Logger.s1:=CONCAT(Logger.s1,DINT_TO_STRING(measures.COSPHI_L1));		Logger.s1:=CONCAT(Logger.s1,';');
Logger.s1:=CONCAT(Logger.s1,DINT_TO_STRING(measures.COSPHI_L2));		Logger.s1:=CONCAT(Logger.s1,';');
Logger.s1:=CONCAT(Logger.s1,DINT_TO_STRING(measures.COSPHI_L3));		Logger.s1:=CONCAT(Logger.s1,';');

Logger.s1:=CONCAT(Logger.s1,BYTE_TO_STRING(SEL(contabilizerMode=THREE_PHASE,1,0)));

ADDSTRING(ADR(Logger.TData), ADR(Logger.s1), Logger.TLen);*)
;
END_ACTION
ACTION checkAlarm:
(*IF(alarmLaunched[1]=0 AND typ_750_494_State.xPhase1_OverCurrentSystem) THEN
	alarmLaunched[1]:=2;
	LogEv(EL_Alarm,EO_ANZ,ID,3, 'xPhase1_OverCurrentSystem');
ELSIF (alarmLaunched[1]=2 AND NOT(typ_750_494_State.xPhase1_OverCurrentSystem) ) THEN
	alarmLaunched[1]:=0;
	LogEv(EL_Log,EO_ANZ,ID,4,'xPhase1_OverCurrentSystem');
END_IF*)

;
END_ACTION
ACTION checkEventsToSignal:
CheckAlarm();
CheckWarning();
CheckStatus();
END_ACTION
ACTION checkStatus:
(*tmpAlarm:=0;
FOR I:=1 TO MAX_alarm DO tmpAlarm:=tmpAlarm+alarmLaunched[i]; END_FOR
IF(tmpAlarm>0) THEN status_Log:=2; END_IF

tmpWarning:=0;
FOR I:=1 TO MAX_WARNING DO tmpWarning:=tmpWarning+warningLaunched[i]; END_FOR
IF(status=0 AND tmpWarning>0) THEN status:=1; END_IF

IF (tmpAlarm =0 AND tmpWarning =0) THEN status:=0; END_IF*)
;
END_ACTION
ACTION checkWarning:
IF(enableWarning = FALSE) THEN RETURN; END_IF

(*IF( warningLaunched[1]=0 AND typ_750_494_State.xGeneralError) THEN
	warningLaunched[1]:=2;
	LogEv(EL_Wrn,EO_ANZ,ID,5, 'xGeneralError');
ELSIF (warningLaunched[1]=2 AND NOT(typ_750_494_State.xGeneralError) ) THEN
	warningLaunched[1]:=0;
	LogEv(EL_Log,EO_ANZ,ID,5,'xGeneralError');
END_IF*)

;
END_ACTION
ACTION convertToClevergyFormat:
	measures.V_L1N := specificData.arVoltage_L_N[1];
	measures.V_L2N := specificData.arVoltage_L_N[2];
	measures.V_L3N := specificData.arVoltage_L_N[3];

	(*n/a*)
	measures.V_L1L2:=0;
	measures.V_L2L3:=0;
	measures.V_L3L1:=0;

	measures.FREQ := specificData.arFrequency*1000;

	measures.I_L1 := specificData.arCurrent[1]*1000;
	measures.I_L2 := specificData.arCurrent[2]*1000;
	measures.I_L3 :=specificData.arCurrent[3]*1000;

	measures.I_L1_Max := specificData.rMaximumCurrentL1*1000;
	measures.I_L2_Max := specificData.rMaximumCurrentL2*1000;
	measures.I_L3_Max := specificData.rMaximumCurrentL3*1000;

	measures.PF_L1 := specificData.arPowerFactorPF[1]*1000;
	measures.PF_L2 := specificData.arPowerFactorPF[2]*1000;
	measures.PF_L3 := specificData.arPowerFactorPF[3]*1000;

	measures.P_3P := specificData.rTotalActivePower*1000;
	measures.P_3P_Avg:=specificData.rAverageTotalActivePower*1000;
	measures.P_3P_Max:=specificData.rMaximumTotalActivePower*1000;

	measures.Q_3P:=specificData.rTotalReactivePower*1000;
	measures.Q_3P_Max:=specificData.rMaximumTotalReactivePower*1000;

	measures.WH_3P:=specificData.rTotalActiveEnergy*10;
	measures.VARH_3P:=specificData.rTotalReactiveEnergy*10;

	(*n/a*)
	measures.COSPHI_L1:=0;
	measures.COSPHI_L2:=0;
	measures.COSPHI_L3:=0;
END_ACTION
ACTION convertToClevergyFormat_OLD:
	measures.V_L1N := REAL_TO_DWORD(specificData.arVoltage_L_N[1]);
	measures.V_L2N := REAL_TO_DWORD(specificData.arVoltage_L_N[2]);
	measures.V_L3N := REAL_TO_DWORD(specificData.arVoltage_L_N[3]);

	(*n/a*)
	measures.V_L1L2:=REAL_TO_DWORD(0);
	measures.V_L2L3:=REAL_TO_DWORD(0);
	measures.V_L3L1:=REAL_TO_DWORD(0);

	measures.FREQ := REAL_TO_DWORD(specificData.arFrequency*1000);

	measures.I_L1 := REAL_TO_DWORD(specificData.arCurrent[1]*1000);
	measures.I_L2 := REAL_TO_DWORD(specificData.arCurrent[2]*1000);
	measures.I_L3 := REAL_TO_DWORD(specificData.arCurrent[3]*1000);

	measures.I_L1_Max := REAL_TO_DWORD(specificData.rMaximumCurrentL1*1000);
	measures.I_L2_Max := REAL_TO_DWORD(specificData.rMaximumCurrentL2*1000);
	measures.I_L3_Max := REAL_TO_DWORD(specificData.rMaximumCurrentL3*1000);

	measures.PF_L1 := REAL_TO_DINT(specificData.arPowerFactorPF[1]*1000);
	measures.PF_L2 := REAL_TO_DINT(specificData.arPowerFactorPF[2]*1000);
	measures.PF_L3 := REAL_TO_DINT(specificData.arPowerFactorPF[3]*1000);

	measures.P_3P := REAL_TO_DINT(specificData.rTotalActivePower);
	measures.P_3P_Avg:=REAL_TO_DINT(specificData.rAverageTotalActivePower);
	measures.P_3P_Max:=REAL_TO_DINT(specificData.rMaximumTotalActivePower);

	measures.Q_3P:=REAL_TO_DINT(specificData.rTotalReactivePower);
	measures.Q_3P_Max:=REAL_TO_DINT(specificData.rMaximumTotalReactivePower);

	measures.WH_3P:=REAL_TO_DINT(specificData.rTotalActiveEnergy*10);
	measures.VARH_3P:=REAL_TO_DINT(specificData.rTotalReactiveEnergy*10);

	(*n/a*)
	measures.COSPHI_L1:=REAL_TO_DINT(0);
	measures.COSPHI_L2:=REAL_TO_DINT(0);
	measures.COSPHI_L3:=REAL_TO_DINT(0);
;
END_ACTION
ACTION getModbusData:
specificData.arFrequency:=modBusConnector.regData[4];

specificData.arVoltage_L_N[1]:=modBusConnector.regData[1];
specificData.arVoltage_L_N[2]:=modBusConnector.regData[2];
specificData.arVoltage_L_N[3]:=modBusConnector.regData[3];

specificData.arCurrent[1]:=modBusConnector.regData[5];
specificData.arCurrent[2]:=modBusConnector.regData[6];
specificData.arCurrent[3]:=modBusConnector.regData[7];

specificData.rTotalActivePower:=modBusConnector.regData[8];
specificData.arActivePower[1]:=modBusConnector.regData[9];
specificData.arActivePower[2]:=modBusConnector.regData[10];
specificData.arActivePower[3]:=modBusConnector.regData[11];

specificData.rTotalReactivePower:=modBusConnector.regData[12];
specificData.arReactivePower[1]:=modBusConnector.regData[13];
specificData.arReactivePower[2]:=modBusConnector.regData[14];
specificData.arReactivePower[3]:=modBusConnector.regData[15];

specificData.rTotalApparentPower:=modBusConnector.regData[16];
specificData.arApparentPower[1]:=modBusConnector.regData[17];
specificData.arApparentPower[2]:=modBusConnector.regData[18];
specificData.arApparentPower[3]:=modBusConnector.regData[19];

specificData.rTotalPowerFactorPF:=modBusConnector.regData[20];
specificData.arPowerFactorPF[1]:=modBusConnector.regData[21];
specificData.arPowerFactorPF[2]:=modBusConnector.regData[22];
specificData.arPowerFactorPF[3]:=modBusConnector.regData[23];

specificData.rTotalActiveEnergy:=modBusConnector.regData[24];

specificData.rTotalReactiveEnergy:=modBusConnector.regData[25];
END_ACTION

(* POU ClevergyBlocks/OBJ_ANZ_INEPRO_PRO380/obj_MODBUS_GENERIC_CONNECTOR, ST *)
FUNCTION_BLOCK obj_MODBUS_GENERIC_CONNECTOR
VAR CONSTANT
		(* States of normal modbus data reading *)
		WAIT_STATE			:	BYTE := 0;
		QUERY_START_CYCLE	: 	BYTE := 1;
		QUERY_MEAS_REQ		:  	BYTE := 2;
		QUERY_MEAS_ANSW	: 	BYTE := 3;
		ERROR_STATE			:	BYTE := 4;
END_VAR
VAR_INPUT
		PARENT_EO_TYPE 		: 	WORD;
		PARENT_EO_ID		:	BYTE;
		Address				:	BYTE;
		TIMING				:	TIME:=t#500ms;

		retryErrMax			:	BYTE := 10;

END_VAR
VAR_IN_OUT
		ModBus		:	obj_MODBUS_ANZ;
END_VAR
VAR_OUTPUT
		Status_Log	:	BYTE;
		Status_Vis	:	DWORD;

		regDescr : ARRAY[1..MODBUS_INEPRO_MAX_REG] OF STRING(20);
		regAddress : ARRAY[1..MODBUS_INEPRO_MAX_REG] OF WORD;
		regQuantity : ARRAY[1..MODBUS_INEPRO_MAX_REG] OF BYTE;
		regValueType : ARRAY[1..MODBUS_INEPRO_MAX_REG] OF en_Modbus_Reg_Type;
		regData: ARRAY[1..MODBUS_INEPRO_MAX_REG] OF REAL;
		regDataWord: ARRAY[1..MODBUS_INEPRO_MAX_REG, 1..2] OF WORD;

END_VAR
VAR
		InitOK		:	BOOL := FALSE;

		(* Modbus State machine variables	*)
		state		:	BYTE;
		last_state		:	BYTE;
		retry		:	BYTE;
		retryErr		:	BYTE;
		ReadTmr		:	TON := (PT:=t#5s);	(* Just to do a first ModBus read at the beginning *)
		fModbusAlr	:	BOOL;

		(* Event check variable	*)
		Alarm		:	FLT_EVENT;
		ModBusAlr	:	FLT_EVENT := (INITEV:=FALSE);
		StatusOK		:	FLT_EVENT := (INITEV:=FALSE);
		AlarmCtr		:	BYTE;
		WarningCtr	:	BYTE;

		fTimeout	:	BOOL;

		currentReg:INT:=1;

		i:INT;
		x:INT;
END_VAR
IF NOT InitOK THEN
	ReadTmr.PT := timing;
	InitOK := TRUE;
	initMapping();
END_IF

(* State machine *)
Stm();

(* Check if an alarm has occured *)
CheckAlarm();

(* Set "Status_Log" according to actual object status	*)
IF AlarmCtr > 0 THEN
	Status_Log := 2;
	Status_Vis := COLOR_RED;
ELSIF WarningCtr > 0 THEN
	Status_Log := 1;
	Status_Vis := COLOR_YELLOW;
ELSE
	Status_Log := 0;

	Status_Vis := COLOR_GREEN;
END_IF
END_FUNCTION_BLOCK
ACTION CheckAlarm:
(*** Verify ModBus error	***)
ModbusAlr(IN:=fModbusAlr);

IF ModbusAlr.EVH THEN
	LogEv(EL_Alarm,PARENT_EO_TYPE,PARENT_EO_ID,2,SEL(ModBus.MB_MASTER.MB_Error<>0,'0','1'));
	AlarmCtr := AlarmCtr + 1;
END_IF

IF ModbusAlr.EVL THEN
	LogEv(EL_Log,PARENT_EO_TYPE,PARENT_EO_ID,1,'');
	AlarmCtr := SEL(AlarmCtr=0, AlarmCtr-1, 0);
END_IF
END_ACTION
ACTION initMapping:
FOR I:=1 TO MODBUS_INEPRO_MAX_REG DO

	IF MODBUS_INEPRO_RegAddress[PARENT_EO_ID,i] <> 0 THEN

		regAddress[i]:=MODBUS_INEPRO_RegAddress[PARENT_EO_ID, i];
		REGDescr[i]:=MODBUS_INEPRO_REGDescr[PARENT_EO_ID, i];
		regQuantity[i]:=MODBUS_INEPRO_regQuantity[PARENT_EO_ID, i];
		regValueType[i]:=MODBUS_INEPRO_regValueType[PARENT_EO_ID, i];

	END_IF

END_FOR
END_ACTION
ACTION Stm:
CASE state OF

	WAIT_STATE:	(* Refresh time manager *)

		ReadTmr(IN:=NOT(ReadTmr.Q));
		IF ReadTmr.Q THEN

			ReadTmr.PT := timing;			(* Refresh timer range *)

			(* Reset state machine variables and counters *)
			retry	:= 0;
			last_state	:= WAIT_STATE;

			(* Start state machine	*)
			state := QUERY_START_CYCLE;

		END_IF

	QUERY_START_CYCLE:
		IF NOT ModBus.MB_Start AND (NOT ModBus.MB_Lock OR retry>0) THEN
			ModBus.MB_Lock := TRUE;

			ModBus.MB_Obj := PARENT_EO_TYPE;
			ModBus.MB_ObjId := PARENT_EO_ID;

			state := QUERY_MEAS_REQ;
		END_IF

	(****			 MEASUREMENTS			  ****)

	QUERY_MEAS_REQ:
		IF NOT ModBus.MB_Start THEN

				IF regAddress[currentReg] <> 0 THEN

					ModBus.MB_Query.SlaveAddress := Address;
					ModBus.MB_Query.FunctionCode := 16#3;
					ModBus.MB_Query.Read_StartAddress :=regAddress[currentReg];
					ModBus.MB_Query.Read_Quantity := regQuantity[currentReg];
					ModBus.MB_Start := TRUE;

					state := QUERY_MEAS_ANSW;

				ELSE

					currentReg:=currentReg+1;

					IF(currentReg<=MODBUS_INEPRO_MAX_REG) THEN

						state := QUERY_MEAS_REQ;

					ELSE

						currentReg:=1;
						fModbusAlr := FALSE;
						retryErr := 0;
						ModBus.MB_Lock := FALSE;
						fTimeout := FALSE;
						state := WAIT_STATE;

					END_IF

				END_IF
		END_IF


	QUERY_MEAS_ANSW:
		IF NOT ModBus.MB_Start THEN
			IF ModBus.MB_MASTER.bInterfaceError<>0 OR ModBus.MB_MASTER.MB_Error<>0 THEN
				last_state := QUERY_MEAS_ANSW;
				state := ERROR_STATE;
			ELSE

				IF (regValueType[currentReg] = VALUE_REAL ) THEN
					regData[currentReg]:=BUILD_REAL_COPY(ModBus.MB_Resp.Data[1],ModBus.MB_Resp.Data[0]);
				END_IF
				IF (regValueType[currentReg] = VALUE_LONG ) THEN
					regDataWord[currentReg,1]:=ModBus.MB_Resp.Data[0];
					regDataWord[currentReg,2]:=ModBus.MB_Resp.Data[1];
				END_IF

				currentReg:=currentReg+1;

				IF(currentReg<=MODBUS_INEPRO_MAX_REG) THEN

					state := QUERY_MEAS_REQ;

				ELSE
					currentReg:=1;
					fModbusAlr := FALSE;
					retryErr := 0;
					ModBus.MB_Lock := FALSE;
					fTimeout := FALSE;
					state := WAIT_STATE;
				END_IF


			END_IF
		END_IF


	ERROR_STATE:	(* Error state *)

		IF retry < 3 THEN
			retry := retry+1;
			state := last_state;

		ELSE
			ModBus.MB_Lock := FALSE;

			(* Verify if slave is dead *)
			IF retryErr < retryErrMaX THEN
				retryErr := retryErr + 1;
			ELSE
				fModbusAlr := TRUE;
			END_IF

			(* Back to wait state *)
			state := WAIT_STATE;

			fTimeout := TRUE;
		END_IF

		IF ModBus.MB_MASTER.MB_Error=MB_TIME_OUT THEN
			state := state;
		END_IF
ELSE
	state := WAIT_STATE;
END_CASE
END_ACTION

(* POU ClevergyBlocks/obj_MODBUS_ANZ, ST *)
FUNCTION_BLOCK obj_MODBUS_ANZ
(* === MODBUS PROTOCOL INTERFACE ===
   v1.1[19/06/15] - Added new VARS allocation and searching
*)
VAR CONSTANT
	VARS_Max	: BYTE := 32;
END_VAR
VAR_INPUT
	(* Settings *)
	ID			: BYTE;
	COM			: BYTE;
	BAUDRATE	: COM_BAUDRATE;
	RS485		: BOOL := FALSE;
	PARITY : COM_PARITY:=PARITY_NO;
	STOP_BITS :COM_STOPBITS:=STOPBITS_2;
	TIME_OUT_TIME : TIME:=t#500ms;

	(* Interface *)
	MB_MASTER	: MODBUS_EXTENDED_MASTER;
	MB_Start	: BOOL;
	MB_Query	: typModbusExtendedQuery;
	MB_Resp		: typModbusResponse;
	MB_Lock		: BOOL;
	MB_Obj		: en_SYS_Objects;
	MB_ObjId	: BYTE;

	(* Variables management *)
	VARS_En		: BOOL := FALSE;
	VARS		: ARRAY [0..VARS_Max] OF typ_MODBUS_VAR_anz;
	VARS_Check	: BOOL;
	VARS_Alarm	: BOOL;

	(* Variables allocation *)
	VAR_Pointer : POINTER TO ARRAY[0..99] OF WORD;
	VAR_Cfg		: POINTER TO typ_MODBUS_VAR_ANZ;
END_VAR
VAR_OUTPUT
	(* Status *)
	Status_Log	: BYTE;
	Status_Vis	: DWORD;
END_VAR
VAR
	sta         : BYTE :=0;
	i			: BYTE;
	j			: BYTE;

	AlarmCOM	: FLT_EVENT;	(* Physical error relative to serial port -> COM	*)
	AlarmMDB	: FLT_EVENT;	(* ModBus error due to communication protocol error	*)

	VarTmr		: TON := (PT:=T#1s);
	VarSta		: BYTE; (* Status *)
	VarCnt		: BYTE; (* Scan counter *)
	VarRetry	: BYTE;
	VarAlarm	: BYTE; (* Last variable with errors *)
END_VAR
MB_MASTER(ENABLE:=TRUE,	ASCII_Mode:=FALSE, bCOM_PORT:=COM, cbCOM_BAUDRATE:=BAUDRATE, cpCOM_PARITY:=PARITY,
		csCOM_STOPBITS:=STOP_BITS,	cbsCOM_BYTESIZE:=BS_8, cfCOM_FLOW_CONTROL:=SEL(RS485,NO_FLOW_CONTROL,HALFDUPLEX),
		tTIME_OUT:=TIME_OUT_TIME,	StartFunction:=MB_Start, ExtQuery:=MB_Query, Response:=MB_Resp);

(* Process variable management *)
IF VARS_En THEN VARS_Process(); END_IF

(* Check status *)
AlarmCOM(IN:=(MB_MASTER.bInterfaceError<>0));
IF AlarmCOM.EVH THEN
	LogEv(SEL(MB_MASTER.bInterfaceError<>3,EL_Wrn,EL_Alarm),EO_MODBUS,ID,1,BYTE_TO_STRING(MB_MASTER.bInterfaceError));
END_IF
IF AlarmCOM.EVL THEN								(* Trigger a fall edge: MODBUS back working *)
	LogEv(EL_Log,EO_MODBUS,ID,2,'MODBUS_OK');
END_IF

(* If VARS not active check if a protocol error has occured (if VARS active this check is already done in "VARS_Process"	*)
IF NOT VARS_En THEN

	AlarmMDB(IN:=(MB_MASTER.MB_Error<>0));
(*	IF AlarmMDB.EVH THEN
		LogEv(EL_Wrn,EO_MODBUS,ID,2,INT_TO_STRING(MB_MASTER.MB_Error));
	END_IF
	IF AlarmMDB.EVL THEN								(* Trigger a fall edge: MODBUS back working *)
		LogEv(EL_Log,EO_MODBUS,ID,2,'MODBUS_OK');
	END_IF
*)
END_IF

(* Log/visu status *)
IF AlarmCOM.IN THEN Status_Log:=2; Status_Vis:=COLOR_RED;
ELSIF Vars_Alarm OR AlarmMDB.IN THEN Status_Log:=1; Status_Vis:=COLOR_YELLOW;
ELSE Status_Log:=0; Status_Vis:=COLOR_GREEN;
END_IF
END_FUNCTION_BLOCK
ACTION VAR_Search:
(* Search VAR with specific pointer if not found return first free VAR
	[Last VAR is not active... used as safe area...] 
*)
j:=VARS_Max;
FOR i := 0 TO VARS_Max-1 DO
	IF VARS[i].Variable=0 AND j>i THEN j:=i; END_IF
	IF VARS[i].Variable=VAR_Pointer THEN
		VAR_Cfg:=ADR(VARS[i]);
		RETURN;
	END_IF
END_FOR
VAR_Cfg:=ADR(VARS[j]);
END_ACTION
ACTION VARS_Process:
(* Update var timers *)
VarTmr(IN:=(NOT VarTmr.Q));
IF VarTmr.Q THEN
	FOR i := 0 TO VARS_Max DO
		IF VARS[i].Refresh_Cnt>0 THEN VARS[i].Refresh_Cnt:=VARS[i].Refresh_Cnt-1; END_IF
	END_FOR
	VARS_Check:=TRUE;
END_IF


(* Process status *)
CASE VarSta OF
	0: (* === Init *)
		VarCnt:=0;
		VarSta:=1;

	1: (* === Wait check signal *)
		IF VARS_Check THEN				(* Decremented "Refresh_Cnt" *)
			VARS_Check:=FALSE;
			VarCnt:=0;
			VarSta:=2;
		END_IF

	2: (* === Check loop *)
		IF NOT (MB_Lock OR MB_Start) THEN
			WHILE VarCnt<=(VARS_Max-1) AND VarSta=2 DO
				(* Check only active vars *)
				IF VARS[VarCnt].Variable<>0 THEN			(* "Variable" is a pointer to word, so if 0 no address *)
					(* Check var auto-refresh on timer checks *)
					IF VARS[VarCnt].Refresh_Time>0 AND VARS[VarCnt].Refresh_Cnt=0 THEN
						VARS[VarCnt].Refresh_Cnt:=VARS[VarCnt].Refresh_Time;
						VarSta:=3;
					END_IF
					(* Check refresh for change or request *)
					CASE VARS[VarCnt].FunCode OF
						5,6,15,16: (* Write functions *)
							IF VARS[VarCnt].Variable_Size=1 THEN
								IF VARS[VarCnt].Variable^[0]<>VARS[VarCnt].Variable_Mirror THEN
									VARS[VarCnt].Variable_Mirror:=VARS[VarCnt].Variable^[0];
									VarSta:=3;
								END_IF
							ELSE
								IF VARS[VarCnt].Variable_Mirror<>0 THEN
									VARS[VarCnt].Variable_Mirror:=0;
									VarSta:=3;
								END_IF
							END_IF
						1,2,3,4: (* Read functions *)
							IF VARS[VarCnt].Variable_Mirror<>0 THEN
								VARS[VarCnt].Variable_Mirror:=0;
								VarSta:=3;
							END_IF
					END_CASE
				END_IF
				(* Process query *)
				IF VarSta=3 THEN
					MB_Lock:=TRUE;
					MB_Query.SlaveAddress:=VARS[VarCnt].SlaveAddress;
					MB_Query.FunctionCode:=VARS[VarCnt].FunCode;
					CASE VARS[VarCnt].FunCode OF
						16#5,16#6,16#F,16#10:
							MB_Query.Read_Quantity:=0;
							MB_Query.Read_StartAddress:=0;
							MB_Query.Write_StartAddress:=VARS[VarCnt].FunAddress;
							MB_Query.Write_Quantity:=VARS[VarCnt].Variable_Size;
							IF VARS[VarCnt].Variable_Size=200 THEN
								COPY_32SWAP16(VARS[VarCnt].Variable, ADR(MB_Query.Write_Data[0]));
							ELSIF VARS[VarCnt].Variable_Size>1 THEN
								MEMCPY(VARS[VarCnt].Variable, ADR(MB_Query.Write_Data[0]), 2*VARS[VarCnt].Variable_Size);
							ELSE
								MB_Query.Write_Data[0]:=VARS[VarCnt].Variable^[0];
							END_IF
						16#1,16#2,16#3,16#4:
							MB_Query.Read_StartAddress:=VARS[VarCnt].FunAddress;
							IF VARS[VarCnt].Variable_Size=200 THEN MB_Query.Read_Quantity:=2; ELSE
							  MB_Query.Read_Quantity:=VARS[VarCnt].Variable_Size;
							END_IF
							MB_Query.Write_StartAddress:=0;
							MB_Query.Write_Quantity:=0;
					END_CASE
					VarRetry:=0;
					MB_Start:=TRUE;
				ELSE
					VarCnt:=VarCnt+1;
				END_IF
			END_WHILE
			(* Check loop completed -> no actions *)
			IF VarSta=2 THEN VarSta:=1; END_IF
		END_IF

	3: (* === Wait & process MB response *)
		IF NOT MB_Start THEN
			IF MB_MASTER.MB_Error=0 THEN
				CASE VARS[VarCnt].FunCode OF
					1,2,3,4:
						IF VARS[VarCnt].Variable_Size=200 THEN
							COPY_32SWAP16(ADR(MB_Resp.Data), VARS[VarCnt].Variable);
						ELSIF VARS[VarCnt].Variable_Size>1 THEN
							MEMCPY(ADR(MB_Resp.Data), VARS[VarCnt].Variable, 2*VARS[VarCnt].Variable_Size);
						ELSE
							VARS[VarCnt].Variable^[0]:=MB_Resp.Data[0];
						END_IF
				END_CASE
				MB_Lock:=FALSE;
				(* Signal error recovery *)
				IF VARS_Alarm=TRUE AND VarCnt=VarAlarm THEN
					LogEv(EL_Wrn,EO_MODBUS,ID,5,'');
					VARS_Alarm:=FALSE;
				END_IF
				(* Next var *)
				VarCnt:=VarCnt+1;
				VarSta:=2;
			ELSE
				IF VarRetry<3 THEN
					VarRetry:=VarRetry+1;
					MB_Start:=TRUE;
				ELSE
					MB_Lock:=FALSE;
					(* Signal error *)
					IF VARS_Alarm=FALSE THEN
						LogEv(EL_Wrn,EO_MODBUS,ID,3,INT_TO_STRING(MB_MASTER.MB_Error));
						VARS_Alarm:=TRUE;
						VarAlarm:=VarCnt-1;
					END_IF
					(* Next var *)
					VarCnt:=VarCnt+1;
					VarSta:=2;
				END_IF
			END_IF
		END_IF

ELSE
	VarSta:=0;
END_CASE
END_ACTION

(* POU Plant_Objects/obj_COMPRESSORE_NEW, ST *)
FUNCTION_BLOCK obj_COMPRESSORE_NEW
VAR CONSTANT

	TimeOutModBus: TON;


END_VAR
VAR_INPUT
	ID			:	BYTE;
	Address		:	BYTE;


	(* Modbus *)
	Refresh_Now	:	BOOL;			(* Richiesta di lettura stato macchina Immediata  *)
	retryErrMax	:	BYTE := 2;

	OnOff		: 	BOOL;

	IndirizzoDaScrivere: WORD;
	DatoDaScrivere: INT;
	ScriviDato: BOOL;
	ScriviCoil: BOOL;

	fWriteAttivazioneComandi:BOOL;


END_VAR
VAR_IN_OUT
	ModBus		:obj_MODBUS;
END_VAR
VAR_OUTPUT
	Run			:	BOOL;

	Status_Log	:	WORD;
	Status_Vis	:	DWORD;
END_VAR
VAR
	(* da diego per gestione stato stringa > 255*)
	temp :STRING(255);
	tempRaw		: ARRAY [0..MAX_SEND_TCP_CLIENT] OF BYTE;
	tempRawLen :DINT;
	longString:STRING(255);

	(* Timer manage switch on/off delay *)
	Delay		: 	TONOF;
	Warning		:	FLT_TAP := (TAP:=100);
	AllarmeCompressore_MB		:	FLT_TAP;

	state		:	INT;
	retry		:	BYTE;
	retryErr	:	BYTE;
	ReadTmr		:	TON := (PT:=T#5s);
	fModbusAlr:BOOL;

	Ctrl_Run: BOOL;


	VerificaFuctionCode: INT;
	VerificaNodoLetto: INT;
	ErroreComuModBus: BOOL;
	IndiceErrore: BYTE;

	MB_BitStato: ARRAY [0..1] OF BOOL;
	MB_RegistriLetti: ARRAY [0..1] OF INT;
	MB_RegistriHoldingLetti: ARRAY [0..260] OF INT;
	MB_BitStatoCoil: ARRAY [0..1] OF BOOL;



	AddressRead: BYTE;
	index: BYTE;
	indexErr: BYTE;





	x: INT;
	moreno1: INT;
	moreno2: INT;
	IndirizzoStart: INT;
	Stop: BOOL;
	start: BOOL;
	StatusControl: ARRAY [0..15] OF BOOL;
END_VAR
(* Call ModBus state machine *)
Stm();

(* Check alarm	*)
CheckAlarm();

(* Seganalzione stato Compressore  *)
IF ErroreComuModBus THEN
		Status_Log:=2; Status_Vis:=16#2020F0;
(*	ELSIF Warning OR Warning2 THEN
		Status_Log:=1; Status_Vis:=16#20F0F0; *)
    ELSE
		Status_Log:=0;
		Status_Vis:=16#006000;
END_IF
END_FUNCTION_BLOCK
ACTION AddLogData:
Logger.s1:=INSERT('&COMPINGRML=',BYTE_TO_STRING(ID),11);
IF ID<10 THEN Logger.s1:=INSERT(Logger.s1,'0',11); END_IF

FOR tempRawLen:=0 TO MAX_SEND_TCP_CLIENT DO
                tempRaw[tempRawLen]:=0;
END_FOR

tempRawLen:=0;


temp:=Logger.s1;
ADDSTRING(ADR(tempRaw), ADR(temp), tempRawLen);

temp:=CONCAT(WORD_TO_STRING(Status_Log),';');
ADDSTRING(ADR(tempRaw), ADR(temp), tempRawLen);


(* Sparo gli ingressi Digitali **)
FOR x:= 0 TO 15 DO
	temp:=CONCAT(SEL(StatusControl[x],'0','1'),';');
	ADDSTRING(ADR(tempRaw), ADR(temp), tempRawLen);
END_FOR

(*

temp:=CONCAT(INT_TO_STRING(MB_RegistriHoldingLetti[1]),';');
ADDSTRING(ADR(tempRaw), ADR(temp), tempRawLen); *)
temp:=CONCAT(INT_TO_STRING(MB_RegistriHoldingLetti[3]),';');
ADDSTRING(ADR(tempRaw), ADR(temp), tempRawLen);
temp:=CONCAT(INT_TO_STRING(MB_RegistriHoldingLetti[4]),';');
ADDSTRING(ADR(tempRaw), ADR(temp), tempRawLen);
temp:=CONCAT(INT_TO_STRING(MB_RegistriHoldingLetti[5]),';');
ADDSTRING(ADR(tempRaw), ADR(temp), tempRawLen);
temp:=CONCAT(INT_TO_STRING(MB_RegistriHoldingLetti[6]),';');
ADDSTRING(ADR(tempRaw), ADR(temp), tempRawLen);
temp:=CONCAT(INT_TO_STRING(MB_RegistriHoldingLetti[11]),';');
ADDSTRING(ADR(tempRaw), ADR(temp), tempRawLen);
temp:=CONCAT(INT_TO_STRING(MB_RegistriHoldingLetti[12]),';');
ADDSTRING(ADR(tempRaw), ADR(temp), tempRawLen);
temp:=CONCAT(INT_TO_STRING(MB_RegistriHoldingLetti[13]),';');
ADDSTRING(ADR(tempRaw), ADR(temp), tempRawLen);
temp:=CONCAT(INT_TO_STRING(MB_RegistriHoldingLetti[14]),';');
ADDSTRING(ADR(tempRaw), ADR(temp), tempRawLen);
temp:=CONCAT(INT_TO_STRING(MB_RegistriHoldingLetti[15]),';');
ADDSTRING(ADR(tempRaw), ADR(temp), tempRawLen);
temp:=CONCAT(INT_TO_STRING(MB_RegistriHoldingLetti[19]),';');
ADDSTRING(ADR(tempRaw), ADR(temp), tempRawLen);
temp:=CONCAT(INT_TO_STRING(MB_RegistriHoldingLetti[20]),';');
ADDSTRING(ADR(tempRaw), ADR(temp), tempRawLen);
temp:=CONCAT(INT_TO_STRING(MB_RegistriHoldingLetti[25]),';');
ADDSTRING(ADR(tempRaw), ADR(temp), tempRawLen);
temp:=CONCAT(INT_TO_STRING(MB_RegistriHoldingLetti[26]),';');
ADDSTRING(ADR(tempRaw), ADR(temp), tempRawLen);
temp:=CONCAT(INT_TO_STRING(MB_RegistriHoldingLetti[27]),';');
ADDSTRING(ADR(tempRaw), ADR(temp), tempRawLen);
temp:=CONCAT(INT_TO_STRING(MB_RegistriHoldingLetti[30]),';');
ADDSTRING(ADR(tempRaw), ADR(temp), tempRawLen);
temp:=CONCAT(INT_TO_STRING(MB_RegistriHoldingLetti[31]),';');
ADDSTRING(ADR(tempRaw), ADR(temp), tempRawLen);
temp:=CONCAT(INT_TO_STRING(MB_RegistriHoldingLetti[64]),';');
ADDSTRING(ADR(tempRaw), ADR(temp), tempRawLen);
temp:=CONCAT(INT_TO_STRING(MB_RegistriHoldingLetti[65]),';');
ADDSTRING(ADR(tempRaw), ADR(temp), tempRawLen);
temp:=CONCAT(INT_TO_STRING(MB_RegistriHoldingLetti[101]),';');
ADDSTRING(ADR(tempRaw), ADR(temp), tempRawLen);
temp:=CONCAT(INT_TO_STRING(MB_RegistriHoldingLetti[112]),';');
ADDSTRING(ADR(tempRaw), ADR(temp), tempRawLen);
temp:=CONCAT(INT_TO_STRING(MB_RegistriHoldingLetti[113]),';');
ADDSTRING(ADR(tempRaw), ADR(temp), tempRawLen);
temp:=CONCAT(INT_TO_STRING(MB_RegistriHoldingLetti[114]),';');
ADDSTRING(ADR(tempRaw), ADR(temp), tempRawLen);
temp:=CONCAT(INT_TO_STRING(MB_RegistriHoldingLetti[115]),';');
ADDSTRING(ADR(tempRaw), ADR(temp), tempRawLen);
temp:=CONCAT(INT_TO_STRING(MB_RegistriHoldingLetti[118]),';');
ADDSTRING(ADR(tempRaw), ADR(temp), tempRawLen);
temp:=CONCAT(INT_TO_STRING(MB_RegistriHoldingLetti[119]),';');
ADDSTRING(ADR(tempRaw), ADR(temp), tempRawLen);
temp:=CONCAT(INT_TO_STRING(MB_RegistriHoldingLetti[121]),';');
ADDSTRING(ADR(tempRaw), ADR(temp), tempRawLen);
temp:=CONCAT(INT_TO_STRING(MB_RegistriHoldingLetti[255]),';');
ADDSTRING(ADR(tempRaw), ADR(temp), tempRawLen);
temp:=(INT_TO_STRING(MB_RegistriHoldingLetti[256]));
ADDSTRING(ADR(tempRaw), ADR(temp), tempRawLen);


ADDSTRING(ADR(Logger.TData), ADR(tempRaw), Logger.TLen);
END_ACTION
ACTION CheckAlarm:
(**** GEstione Log ad Evento *****)




	AllarmeCompressore_MB(IN:=MB_RegistriHoldingLetti[1].6 );

	IF AllarmeCompressore_MB.EVH THEN
		LogEv(EL_Alarm,EO_COMPINGRML,ID,1,CONCAT ('AllarmeAttivo_n.', INT_TO_STRING(MB_RegistriHoldingLetti[255])));
	END_IF

	IF AllarmeCompressore_MB.EVL THEN
		LogEv(EL_Log,EO_COMPINGRML,ID,2,CONCAT ('AllarmeRientrato_n.', INT_TO_STRING(MB_RegistriHoldingLetti[255])));
	END_IF
END_ACTION
ACTION Stm:
CASE state OF
	0:	(* Refresh time manager *)
		ReadTmr(IN:=NOT ReadTmr.Q);
		(*A tempo interrogo il nodo sempre che non ci sia qualcuno che lo sta interrogando in quel momento *)

		IF (ReadTmr.Q AND NodoDaInterrogareCompressoreNuovo=Address ) OR Refresh_Now AND NOT InibiscoModbusCompressoreNuovo THEN
			state := 10;
			ReadTmr.PT := T#100ms;  (* moreno *)
			Refresh_Now := FALSE;
			InibiscoModbusCompressoreNuovo := TRUE;
		END_IF

	(**** Leggo le Analogiche a Disposzione  ****)

	10:	(* richiedo lettura Holding Registere   *)

		Modbus.MB_Query.SlaveAddress := Address;
		Modbus.MB_Query.FunctionCode := 3;
		IndirizzoStart:=1;
		ModBus.MB_Query.Read_StartAddress :=IndirizzoStart - 1 ;
		ModBus.MB_Query.Read_Quantity := 19;(*19;*)
		ModBus.MB_Start := TRUE;
		state := 20;

	20:	(* Risposta all'interrogazione *)
		IF NOT ModBus.MB_Start   THEN
			VerificaFuctionCode:=ModBus.MB_Resp.FunctionCode;
			VerificaNodoLetto:=ModBus.MB_Resp.SlaveAddress;

			IF ModBus.MB_MASTER.MB_Error<>0 THEN
				state := 300;
			ELSE
				FOR x:=0 TO ModBus.MB_Query.Read_Quantity DO
					MB_RegistriHoldingLetti[x+IndirizzoStart] := ModBus.MB_Resp.Data[x];   	(* Vedi tabella *)
				END_FOR

				(* trasforo la wordo in singoli 16 bit *)

					StatusControl[0]:= MB_RegistriHoldingLetti[IndirizzoStart].0;   	(* Vedi tabella *)
					StatusControl[1]:= MB_RegistriHoldingLetti[IndirizzoStart].1;   	(* Vedi tabella *)
					StatusControl[2]:= MB_RegistriHoldingLetti[IndirizzoStart].2;   	(* Vedi tabella *)
					StatusControl[3]:= MB_RegistriHoldingLetti[IndirizzoStart].3;   	(* Vedi tabella *)
					StatusControl[4]:= MB_RegistriHoldingLetti[IndirizzoStart].4;   	(* Vedi tabella *)
					StatusControl[5]:= MB_RegistriHoldingLetti[IndirizzoStart].5;   	(* Vedi tabella *)
					StatusControl[6]:= MB_RegistriHoldingLetti[IndirizzoStart].6;   	(* Vedi tabella *)
					StatusControl[7]:= MB_RegistriHoldingLetti[IndirizzoStart].7;   	(* Vedi tabella *)
					StatusControl[8]:= MB_RegistriHoldingLetti[IndirizzoStart].8;   	(* Vedi tabella *)
					StatusControl[9]:= MB_RegistriHoldingLetti[IndirizzoStart].9;   	(* Vedi tabella *)
					StatusControl[10]:= MB_RegistriHoldingLetti[IndirizzoStart].10;   	(* Vedi tabella *)
					StatusControl[11]:= MB_RegistriHoldingLetti[IndirizzoStart].11;   	(* Vedi tabella *)
					StatusControl[12]:= MB_RegistriHoldingLetti[IndirizzoStart].12;   	(* Vedi tabella *)
					StatusControl[13]:= MB_RegistriHoldingLetti[IndirizzoStart].13;   	(* Vedi tabella *)
					StatusControl[14]:= MB_RegistriHoldingLetti[IndirizzoStart].14;   	(* Vedi tabella *)
					StatusControl[15]:= MB_RegistriHoldingLetti[IndirizzoStart].15;   	(* Vedi tabella *)





				IndirizzoStart:=20;
				ModBus.MB_Query.Read_StartAddress :=IndirizzoStart - 1 ;
				ModBus.MB_Query.Read_Quantity := 19;
				ModBus.MB_Start := TRUE;

				state := 30;
			END_IF
		END_IF

	30: (* Rispota Altri paramenti *)
		IF NOT ModBus.MB_Start  THEN

			IF ModBus.MB_MASTER.MB_Error<>0 THEN
				state := 300;
			ELSE

				FOR x:=0 TO ModBus.MB_Query.Read_Quantity DO
					MB_RegistriHoldingLetti[x+IndirizzoStart] := ModBus.MB_Resp.Data[x];   	(* Vedi tabella *)
				END_FOR

				IndirizzoStart:=40;
				ModBus.MB_Query.Read_StartAddress :=IndirizzoStart - 1 ;
				ModBus.MB_Query.Read_Quantity := 19;
				ModBus.MB_Start := TRUE;

				state := 35;
			END_IF
		END_IF
	35: (* Rispota Altri paramenti *)
		IF NOT ModBus.MB_Start  THEN

			IF ModBus.MB_MASTER.MB_Error<>0 THEN
				state := 300;
			ELSE

				FOR x:=0 TO ModBus.MB_Query.Read_Quantity DO
					MB_RegistriHoldingLetti[x+IndirizzoStart] := ModBus.MB_Resp.Data[x];   	(* Vedi tabella *)
				END_FOR

				IndirizzoStart:=64;
				ModBus.MB_Query.Read_StartAddress :=IndirizzoStart - 1 ;
				ModBus.MB_Query.Read_Quantity := 6;
				ModBus.MB_Start := TRUE;

				state := 40;
			END_IF
		END_IF
	40: (* Rispota Altri paramenti *)
		IF NOT ModBus.MB_Start  THEN

			IF ModBus.MB_MASTER.MB_Error<>0 THEN
				state := 300;
			ELSE

				FOR x:=0 TO ModBus.MB_Query.Read_Quantity DO
					MB_RegistriHoldingLetti[x+IndirizzoStart] := ModBus.MB_Resp.Data[x];   	(* Vedi tabella *)
				END_FOR

				IndirizzoStart:=90;
				ModBus.MB_Query.Read_StartAddress :=IndirizzoStart - 1 ;
				ModBus.MB_Start := TRUE;

				state := 45;
			END_IF
		END_IF

	45: (* Rispota Altri paramenti *)
		IF NOT ModBus.MB_Start  THEN

			IF ModBus.MB_MASTER.MB_Error<>0 THEN
				state := 300;
			ELSE
				FOR x:=0 TO ModBus.MB_Query.Read_Quantity DO
					MB_RegistriHoldingLetti[x+IndirizzoStart] := ModBus.MB_Resp.Data[x];   	(* Vedi tabella *)
				END_FOR

				IndirizzoStart:=110;
				ModBus.MB_Query.Read_StartAddress :=IndirizzoStart - 1 ;
				ModBus.MB_Query.Read_Quantity := 19;
				ModBus.MB_Start := TRUE;

				state := 50;
			END_IF
		END_IF


	50: (* Rispota Altri paramenti *)
		IF NOT ModBus.MB_Start  THEN

			IF ModBus.MB_MASTER.MB_Error<>0 THEN
				state := 300;
			ELSE
				FOR x:=0 TO ModBus.MB_Query.Read_Quantity DO
					MB_RegistriHoldingLetti[x+IndirizzoStart] := ModBus.MB_Resp.Data[x];   	(* Vedi tabella *)
				END_FOR

				IndirizzoStart:=130;
				ModBus.MB_Query.Read_StartAddress :=IndirizzoStart - 1 ;
				ModBus.MB_Query.Read_Quantity := 5;
				ModBus.MB_Start := TRUE;


				state := 55;
			END_IF
		END_IF

	55: (* Rispota Altri paramenti *)
		IF NOT ModBus.MB_Start  THEN

			IF ModBus.MB_MASTER.MB_Error<>0 THEN
				state := 300;
			ELSE
				FOR x:=0 TO ModBus.MB_Query.Read_Quantity DO
					MB_RegistriHoldingLetti[x+IndirizzoStart] := ModBus.MB_Resp.Data[x];   	(* Vedi tabella *)
				END_FOR

				IndirizzoStart:=240;
				ModBus.MB_Query.Read_StartAddress :=IndirizzoStart - 1 ;
				ModBus.MB_Query.Read_Quantity := 3;
				ModBus.MB_Start := TRUE;

				state := 60;
			END_IF
		END_IF

	60: (* Rispota Altri paramenti *)
		IF NOT ModBus.MB_Start  THEN

			IF ModBus.MB_MASTER.MB_Error<>0 THEN
				state := 300;
			ELSE
				FOR x:=0 TO ModBus.MB_Query.Read_Quantity DO
					MB_RegistriHoldingLetti[x+IndirizzoStart] := ModBus.MB_Resp.Data[x];   	(* Vedi tabella *)
				END_FOR

				state :=290;
			END_IF
		END_IF


		290:    (* Scrittura BOOL - COIL o WORD *)
		IF NOT ModBus.MB_Start THEN
			IF ModBus.MB_MASTER.MB_Error<>0 THEN (*OR ModBus.MB_MASTER.MB_Error<>0 THEN*)
				state := 300;
			ELSE
				IF ScriviDato THEN
					IF ScriviCoil THEN
						Modbus.MB_Query.FunctionCode := 5;
					ELSE
						Modbus.MB_Query.FunctionCode := 6;
					END_IF
					Modbus.MB_Query.SlaveAddress := Address;
					ModBus.MB_Query.Write_StartAddress := IndirizzoDaScrivere-1;
					ModBus.MB_Query.Write_Quantity :=1;

					IF Stop THEN
								 DatoDaScrivere:=MB_RegistriHoldingLetti[IndirizzoDaScrivere];
	  							 DatoDaScrivere.0:=TRUE;
  							        DatoDaScrivere.1:=FALSE;
					END_IF
					IF start THEN
								 DatoDaScrivere:=MB_RegistriHoldingLetti[IndirizzoDaScrivere];
	  							 DatoDaScrivere.0:=TRUE;
  							        DatoDaScrivere.1:=TRUE;
					END_IF


					ModBus.MB_Query.Write_Data[0] := DatoDaScrivere;
					ModBus.MB_Start := TRUE;
						IF ScriviCoil THEN
							IF 	MB_BitStato[IndirizzoDaScrivere]=WORD_TO_BOOL(DatoDaScrivere-1) THEN
								ScriviDato:=FALSE;
							END_IF
						ELSE
							IF 	MB_RegistriHoldingLetti[IndirizzoDaScrivere]=DatoDaScrivere THEN
								ScriviDato:=FALSE;
							END_IF
						END_IF
					state := 295;
				ELSE
					state := 295;
				END_IF
			END_IF
		END_IF




		295:
		IF NOT ModBus.MB_Start THEN
			IF ModBus.MB_MASTER.MB_Error<>0 THEN (*OR ModBus.MB_MASTER.MB_Error<>0 THEN*)
				state := 300;
			ELSE
				IF fModbusAlr THEN fModbusAlr := FALSE; END_IF
				NodoDaInterrogareCompressoreNuovo:=Address+1;
				InibiscoModbusCompressoreNuovo:=FALSE;
				retryErr := 0;
				retry := 0;
				state := 0;
					IF fModbusAlr=FALSE AND ErroreComuModBus=TRUE THEN
						LogEv(EL_Log,EO_COMPINGRML,ID,62,'ComunicazioneModBus_OK');
						ErroreComuModBus := FALSE;
				(*	WarningCtr := SEL(WarningCtr=0, WarningCtr-1, 0); *)
					END_IF
			END_IF


		END_IF




	(**** CHECK MODBUS ERROR ****)
	300: 	(* Release MODBUS *)
			InibiscoModbusCompressoreNuovo:=FALSE;
			(* Retries *)
			retry:=retry+1;
			IF retry>3 THEN
				retry:=0;

				(* Verify if slave is dead *)
				IF retryErr < retryErrMaX THEN
					retryErr := retryErr + 1;
				ELSE
					fModbusAlr := TRUE;
					(* Verify ModBus error	*)

					IF fModbusAlr AND ErroreComuModBus=FALSE THEN
						LogEv(EL_Alarm,EO_COMPINGRML,ID,61,CONCAT('ErroreModbus_',INT_TO_STRING(ModBus.MB_MASTER.MB_Error)));
						ErroreComuModBus := TRUE;
					END_IF
				END_IF

				END_IF
			Refresh_Now := FALSE;
			NodoDaInterrogareCompressoreNuovo:=Address+1;
			state:=0;
END_CASE




(* Controllo Time Out Ciclo ModBus *)

TimeOutModBus(In:=state<>0,PT:=t#30s);
IF TimeOutModBus.Q THEN
	State:=0;
	Refresh_Now:=TRUE;  (* Rilancio la lettura del nodo *)
	IF MODBUS.MB_Lock=TRUE THEN MODBUS.MB_Lock:=FALSE;END_IF
	IF InibiscoModbusCompressoreNuovo=TRUE THEN InibiscoModbusCompressoreNuovo:=FALSE;END_IF
	NodoDaInterrogareCompressoreNuovo:=Address+1;

END_IF
END_ACTION

(* POU Plant_Objects/obj_MODBUS, ST *)
FUNCTION_BLOCK obj_MODBUS
(* === MODBUS PROTOCOL INTERFACE ===
   v1.1[19/06/15] - Added new VARS allocation and searching
*)
VAR CONSTANT
	VARS_Max	: BYTE := 32;
END_VAR
VAR_INPUT
	(* Settings *)
	ID			: BYTE;
	COM			: BYTE;
	BAUDRATE	: COM_BAUDRATE;
	RS485		: BOOL := FALSE;

	N_STOPBits	:BYTE:=1;

	(* Interface *)
	MB_MASTER	: MODBUS_EXTENDED_MASTER;
	MB_Start	: BOOL;
	MB_Query	: typModbusExtendedQuery;
	MB_Resp		: typModbusResponse;
	MB_Lock		: BOOL;
	MB_timeOut	: TIME := t#500ms;

	(* Variables management *)
	VARS_En		: BOOL;
	VARS		: ARRAY [0..VARS_Max] OF typ_MODBUS_VAR;
	VARS_Check	: BOOL;
	VARS_Alarm	: BOOL;

	(* Variables allocation *)
	VAR_Pointer : POINTER TO ARRAY[0..99] OF WORD;
	VAR_Cfg		: POINTER TO typ_MODBUS_VAR;
END_VAR
VAR_OUTPUT
	(* Status *)
	Status_Log	: BYTE;
	Status_Vis	: DWORD;
END_VAR
VAR
	sta         : BYTE :=0;
	i			: BYTE;
	j			: BYTE;
	Alarm		: FLT_EVENT;
	
	VarTmr		: TON := (PT:=T#1s);
	VarSta		: BYTE; (* Status *)
	VarCnt		: BYTE; (* Scan counter *)
	VarRetry	: BYTE;
	VarAlarm	: BYTE; (* Last variable with errors *)
END_VAR
IF N_STOPBits=1 THEN MB_MASTER.csCOM_STOPBITS:=STOPBITS_1;END_IF
IF N_STOPBits=2 THEN MB_MASTER.csCOM_STOPBITS:=STOPBITS_2;END_IF

MB_MASTER(ENABLE:=TRUE,	ASCII_Mode:=FALSE, bCOM_PORT:=COM, cbCOM_BAUDRATE:=BAUDRATE, cpCOM_PARITY:=PARITY_NO,
		cbsCOM_BYTESIZE:=BS_8, cfCOM_FLOW_CONTROL:=SEL(RS485,NO_FLOW_CONTROL,HALFDUPLEX),
		tTIME_OUT:=MB_timeOut,	StartFunction:=MB_Start, ExtQuery:=MB_Query, Response:=MB_Resp);

(* Process variable management *)
IF VARS_En THEN VARS_Process(); END_IF

(* Check status *)
Alarm(IN:=(MB_MASTER.bInterfaceError<>0));
IF Alarm.EVH THEN
	LogEv(SEL(MB_MASTER.bInterfaceError<>3,EL_Wrn,EL_Alarm),EO_MODBUS,ID,1,BYTE_TO_STRING(MB_MASTER.bInterfaceError));
END_IF
IF Alarm.EVL THEN								(* Trigger a fall edge: MODBUS back working *)
	LogEv(EL_Log,EO_MODBUS,ID,2,'MODBUS_OK');
END_IF

(* Log/visu status *)
   IF Alarm.IN   THEN Status_Log:=2; Status_Vis:=COLOR_RED;
ELSIF Vars_Alarm THEN Status_Log:=1; Status_Vis:=COLOR_YELLOW;
  				 ELSE Status_Log:=0; Status_Vis:=COLOR_GREEN;
END_IF
END_FUNCTION_BLOCK
ACTION VAR_Search:
(* Search VAR with specific pointer if not found return first free VAR
	[Last VAR is not active... used as safe area...] 
*)
j:=VARS_Max;
FOR i := 0 TO VARS_Max-1 DO
	IF VARS[i].Variable=0 AND j>i THEN j:=i; END_IF
	IF VARS[i].Variable=VAR_Pointer THEN
		VAR_Cfg:=ADR(VARS[i]);
		RETURN;
	END_IF
END_FOR
VAR_Cfg:=ADR(VARS[j]);
END_ACTION
ACTION VARS_Process:
(* Update var timers *)
VarTmr(IN:=(NOT VarTmr.Q));
IF VarTmr.Q THEN
	FOR i := 0 TO VARS_Max DO
		IF VARS[i].Refresh_Cnt>0 THEN VARS[i].Refresh_Cnt:=VARS[i].Refresh_Cnt-1; END_IF
	END_FOR
	VARS_Check:=TRUE;
END_IF


(* Process status *)
CASE VarSta OF
	0: (* === Init *)
		VarCnt:=0;
		VarSta:=1;

	1: (* === Wait check signal *)
		IF VARS_Check THEN				(* Decremented "Refresh_Cnt" *)
			VARS_Check:=FALSE;
			VarCnt:=0;
			VarSta:=2;
		END_IF

	2: (* === Check loop *)
		IF NOT (MB_Lock OR MB_Start) THEN
			WHILE VarCnt<=(VARS_Max-1) AND VarSta=2 DO
				(* Check only active vars *)
				IF VARS[VarCnt].Variable<>0 THEN			(* "Variable" is a pointer to word, so if 0 no address *)
					(* Check var auto-refresh on timer checks *)
					IF VARS[VarCnt].Refresh_Time>0 AND VARS[VarCnt].Refresh_Cnt=0 THEN
						VARS[VarCnt].Refresh_Cnt:=VARS[VarCnt].Refresh_Time;
						VarSta:=3;
					END_IF
					(* Check refresh for change or request *)
					CASE VARS[VarCnt].FunCode OF
						5,6,15,16: (* Write functions *)
							IF VARS[VarCnt].Variable_Size=1 THEN
								IF VARS[VarCnt].Variable^<>VARS[VarCnt].Variable_Mirror THEN
									VARS[VarCnt].Variable_Mirror:=VARS[VarCnt].Variable^;
									VarSta:=3;
								END_IF
							ELSE
								IF VARS[VarCnt].Variable_Mirror<>0 THEN
									VARS[VarCnt].Variable_Mirror:=0;
									VarSta:=3;
								END_IF
							END_IF
						1,2,3,4: (* Read functions *)
							IF VARS[VarCnt].Variable_Mirror<>0 THEN
								VARS[VarCnt].Variable_Mirror:=0;
								VarSta:=3;
							END_IF
					END_CASE
				END_IF
				(* Process query *)
				IF VarSta=3 THEN
					MB_Lock:=TRUE;
					MB_Query.SlaveAddress:=VARS[VarCnt].SlaveAddress;
					MB_Query.FunctionCode:=VARS[VarCnt].FunCode;
					CASE VARS[VarCnt].FunCode OF
						16#5,16#6,16#F,16#10:
							MB_Query.Read_Quantity:=0;
							MB_Query.Read_StartAddress:=0;
							MB_Query.Write_StartAddress:=VARS[VarCnt].FunAddress;
							MB_Query.Write_Quantity:=VARS[VarCnt].Variable_Size;
							IF VARS[VarCnt].Variable_Size=200 THEN
								COPY_32SWAP16(VARS[VarCnt].Variable, ADR(MB_Query.Write_Data[0]));
							ELSIF VARS[VarCnt].Variable_Size>1 THEN
								MEMCPY(VARS[VarCnt].Variable, ADR(MB_Query.Write_Data[0]), 2*VARS[VarCnt].Variable_Size);
							ELSE
								MB_Query.Write_Data[0]:=VARS[VarCnt].Variable^;
							END_IF
						16#1,16#2,16#3,16#4:
							MB_Query.Read_StartAddress:=VARS[VarCnt].FunAddress;
							IF VARS[VarCnt].Variable_Size=200 THEN MB_Query.Read_Quantity:=2; ELSE
							  MB_Query.Read_Quantity:=VARS[VarCnt].Variable_Size;
							END_IF
							MB_Query.Write_StartAddress:=0;
							MB_Query.Write_Quantity:=0;
					END_CASE
					VarRetry:=0;
					MB_Start:=TRUE;
				ELSE
					VarCnt:=VarCnt+1;
				END_IF
			END_WHILE
			(* Check loop completed -> no actions *)
			IF VarSta=2 THEN VarSta:=1; END_IF
		END_IF

	3: (* === Wait & process MB response *)
		IF NOT MB_Start THEN
			IF MB_MASTER.MB_Error=0 THEN
				CASE VARS[VarCnt].FunCode OF
					1,2,3,4:
						IF VARS[VarCnt].Variable_Size=200 THEN
							COPY_32SWAP16(ADR(MB_Resp.Data), VARS[VarCnt].Variable);
						ELSIF VARS[VarCnt].Variable_Size>1 THEN
							MEMCPY(ADR(MB_Resp.Data), VARS[VarCnt].Variable, 2*VARS[VarCnt].Variable_Size);
						ELSE
							VARS[VarCnt].Variable^:=MB_Resp.Data[0];
						END_IF
				END_CASE
				MB_Lock:=FALSE;
				(* Signal error recovery *)
				IF VARS_Alarm=TRUE AND VarCnt=VarAlarm THEN
					LogEv(EL_Wrn,EO_MODBUS,ID,5,'');
					VARS_Alarm:=FALSE;
				END_IF
				(* Next var *)
				VarCnt:=VarCnt+1;
				VarSta:=2;
			ELSE
				IF VarRetry<3 THEN
					VarRetry:=VarRetry+1;
					MB_Start:=TRUE;
				ELSE
					MB_Lock:=FALSE;
					(* Signal error *)
					IF VARS_Alarm=FALSE THEN
						LogEv(EL_Wrn,EO_MODBUS,ID,3,INT_TO_STRING(MB_MASTER.MB_Error));
						VARS_Alarm:=TRUE;
						VarAlarm:=VarCnt-1;
					END_IF
					(* Next var *)
					VarCnt:=VarCnt+1;
					VarSta:=2;
				END_IF
			END_IF
		END_IF

ELSE
	VarSta:=0;
END_CASE
END_ACTION

(* POU Utils Functions/TONOF, ST *)
FUNCTION_BLOCK TONOF
VAR_INPUT
	IN		: BOOL;
	PT_ON	: TIME; (* time to pass, before OUT is set *)
	PT_OF	: TIME; (* time to pass, before OUT is reset *)
END_VAR
VAR_OUTPUT
	OUT		: BOOL;
END_VAR
VAR
	timer	: TON;
END_VAR
IF IN<>OUT THEN
	timer(IN:=TRUE,PT:=SEL(IN,PT_OF,PT_ON));
	IF timer.Q THEN OUT:=IN; END_IF
ELSE
	timer(IN:=FALSE);
END_IF
END_FUNCTION_BLOCK

(* POU Plant_Objects/obj_COMPRESSORE_OLD, ST *)
FUNCTION_BLOCK obj_COMPRESSORE_OLD
VAR CONSTANT

	TimeOutModBus: TON;

END_VAR
VAR_INPUT
	ID			:	BYTE;
	Address		:	BYTE;


	(* Modbus *)
	Refresh_Now	:	BOOL;			(* Richiesta di lettura stato macchina Immediata  *)
	retryErrMax	:	BYTE := 2;

	OnOff		: 	BOOL;

	IndirizzoDaScrivere: WORD;
	DatoDaScrivere: INT;
	ScriviDato: BOOL;
	ScriviCoil: BOOL;

	fWriteAttivazioneComandi:BOOL;


END_VAR
VAR_IN_OUT
	ModBus		:obj_MODBUS;
END_VAR
VAR_OUTPUT
	Run			:	BOOL;

	Status_Log	:	WORD;
	Status_Vis	:	DWORD;
END_VAR
VAR
	(* da diego per gestione stato stringa > 255*)
	temp :STRING(255);
	tempRaw		: ARRAY [0..MAX_SEND_TCP_CLIENT] OF BYTE;
	tempRawLen :DINT;
	longString:STRING(255);

	(* Timer manage switch on/off delay *)
	Delay		: 	TONOF;
	Warning		:	FLT_TAP := (TAP:=100);
	AllarmeCompressore_MB		:	FLT_TAP;

	state		:	INT;
	retry		:	BYTE;
	retryErr	:	BYTE;
	ReadTmr		:	TON := (PT:=T#5s);
	fModbusAlr:BOOL;

	Ctrl_Run: BOOL;


	VerificaFuctionCode: INT;
	VerificaNodoLetto: INT;
	ErroreComuModBus: BOOL;
	IndiceErrore: BYTE;

	MB_BitStato: ARRAY [0..1] OF BOOL;
	MB_RegistriLetti: ARRAY [0..1] OF INT;
	MB_RegistriHoldingLetti: ARRAY [0..400] OF INT;
	MB_BitStatoCoil: ARRAY [0..1] OF BOOL;



	AddressRead: BYTE;
	index: BYTE;
	indexErr: BYTE;

	x: INT;
	IndirizzoStart: INT;
	Stop: BOOL;
	start: BOOL;
	StatusControl: ARRAY [0..15] OF BOOL;


END_VAR
(* Call ModBus state machine *)
Stm();

(* Check alarm	*)
CheckAlarm();

(* Seganalzione stato Compressore  *)
IF ErroreComuModBus THEN
		Status_Log:=2; Status_Vis:=16#2020F0;
(*	ELSIF Warning OR Warning2 THEN
		Status_Log:=1; Status_Vis:=16#20F0F0; *)
    ELSE
		Status_Log:=0;
		Status_Vis:=16#006000;
END_IF
END_FUNCTION_BLOCK
ACTION AddLogData:
Logger.s1:=INSERT('&COMPINGRR=',BYTE_TO_STRING(ID),10);
IF ID<10 THEN Logger.s1:=INSERT(Logger.s1,'0',10); END_IF

FOR tempRawLen:=0 TO MAX_SEND_TCP_CLIENT DO
                tempRaw[tempRawLen]:=0;
END_FOR

tempRawLen:=0;


temp:=Logger.s1;
ADDSTRING(ADR(tempRaw), ADR(temp), tempRawLen);


(* Sparo gli ingressi Digitali **)
FOR x:= 0 TO 15 DO
	temp:=CONCAT(SEL(StatusControl[x],'0','1'),';');
	ADDSTRING(ADR(tempRaw), ADR(temp), tempRawLen);
END_FOR

(*

temp:=CONCAT(INT_TO_STRING(MB_RegistriHoldingLetti[1]),';');
ADDSTRING(ADR(tempRaw), ADR(temp), tempRawLen); *)
temp:=CONCAT(INT_TO_STRING(MB_RegistriHoldingLetti[1]),';');
ADDSTRING(ADR(tempRaw), ADR(temp), tempRawLen);
temp:=CONCAT(INT_TO_STRING(MB_RegistriHoldingLetti[3]),';');
ADDSTRING(ADR(tempRaw), ADR(temp), tempRawLen);
temp:=CONCAT(INT_TO_STRING(MB_RegistriHoldingLetti[4]),';');
ADDSTRING(ADR(tempRaw), ADR(temp), tempRawLen);
temp:=CONCAT(INT_TO_STRING(MB_RegistriHoldingLetti[5]),';');
ADDSTRING(ADR(tempRaw), ADR(temp), tempRawLen);
temp:=CONCAT(INT_TO_STRING(MB_RegistriHoldingLetti[6]),';');
ADDSTRING(ADR(tempRaw), ADR(temp), tempRawLen);
temp:=CONCAT(INT_TO_STRING(MB_RegistriHoldingLetti[7]),';');
ADDSTRING(ADR(tempRaw), ADR(temp), tempRawLen);
temp:=CONCAT(INT_TO_STRING(MB_RegistriHoldingLetti[8]),';');
ADDSTRING(ADR(tempRaw), ADR(temp), tempRawLen);
temp:=CONCAT(INT_TO_STRING(MB_RegistriHoldingLetti[9]),';');
ADDSTRING(ADR(tempRaw), ADR(temp), tempRawLen);
temp:=CONCAT(INT_TO_STRING(MB_RegistriHoldingLetti[10]),';');
ADDSTRING(ADR(tempRaw), ADR(temp), tempRawLen);
temp:=CONCAT(INT_TO_STRING(MB_RegistriHoldingLetti[20]),';');
ADDSTRING(ADR(tempRaw), ADR(temp), tempRawLen);
temp:=CONCAT(INT_TO_STRING(MB_RegistriHoldingLetti[64]),';');
ADDSTRING(ADR(tempRaw), ADR(temp), tempRawLen);
temp:=CONCAT(INT_TO_STRING(MB_RegistriHoldingLetti[65]),';');
ADDSTRING(ADR(tempRaw), ADR(temp), tempRawLen);
temp:=CONCAT(INT_TO_STRING(MB_RegistriHoldingLetti[66]),';');
ADDSTRING(ADR(tempRaw), ADR(temp), tempRawLen);
temp:=CONCAT(INT_TO_STRING(MB_RegistriHoldingLetti[67]),';');
ADDSTRING(ADR(tempRaw), ADR(temp), tempRawLen);
temp:=CONCAT(INT_TO_STRING(MB_RegistriHoldingLetti[98]),';');
ADDSTRING(ADR(tempRaw), ADR(temp), tempRawLen);
temp:=CONCAT(INT_TO_STRING(MB_RegistriHoldingLetti[103]),';');
ADDSTRING(ADR(tempRaw), ADR(temp), tempRawLen);
temp:=CONCAT(INT_TO_STRING(MB_RegistriHoldingLetti[112]),';');
ADDSTRING(ADR(tempRaw), ADR(temp), tempRawLen);
temp:=CONCAT(INT_TO_STRING(MB_RegistriHoldingLetti[113]),';');
ADDSTRING(ADR(tempRaw), ADR(temp), tempRawLen);
temp:=CONCAT(INT_TO_STRING(MB_RegistriHoldingLetti[114]),';');
ADDSTRING(ADR(tempRaw), ADR(temp), tempRawLen);
temp:=CONCAT(INT_TO_STRING(MB_RegistriHoldingLetti[116]),';');
ADDSTRING(ADR(tempRaw), ADR(temp), tempRawLen);
temp:=CONCAT(INT_TO_STRING(MB_RegistriHoldingLetti[117]),';');
ADDSTRING(ADR(tempRaw), ADR(temp), tempRawLen);
temp:=CONCAT(INT_TO_STRING(MB_RegistriHoldingLetti[123]),';');
ADDSTRING(ADR(tempRaw), ADR(temp), tempRawLen);
temp:=CONCAT(INT_TO_STRING(MB_RegistriHoldingLetti[125]),';');
ADDSTRING(ADR(tempRaw), ADR(temp), tempRawLen);
temp:=CONCAT(INT_TO_STRING(MB_RegistriHoldingLetti[130]),';');
ADDSTRING(ADR(tempRaw), ADR(temp), tempRawLen);
temp:=CONCAT(INT_TO_STRING(MB_RegistriHoldingLetti[255]),';');
ADDSTRING(ADR(tempRaw), ADR(temp), tempRawLen);
temp:=CONCAT(INT_TO_STRING(MB_RegistriHoldingLetti[256]),';');
ADDSTRING(ADR(tempRaw), ADR(temp), tempRawLen);
temp:=CONCAT(INT_TO_STRING(MB_RegistriHoldingLetti[257]),';');
ADDSTRING(ADR(tempRaw), ADR(temp), tempRawLen);
temp:=CONCAT(INT_TO_STRING(MB_RegistriHoldingLetti[258]),';');
ADDSTRING(ADR(tempRaw), ADR(temp), tempRawLen);
temp:=CONCAT(INT_TO_STRING(MB_RegistriHoldingLetti[259]),';');
ADDSTRING(ADR(tempRaw), ADR(temp), tempRawLen);
temp:=CONCAT(INT_TO_STRING(MB_RegistriHoldingLetti[260]),';');
ADDSTRING(ADR(tempRaw), ADR(temp), tempRawLen);
temp:=CONCAT(INT_TO_STRING(MB_RegistriHoldingLetti[261]),';');
ADDSTRING(ADR(tempRaw), ADR(temp), tempRawLen);
temp:=CONCAT(INT_TO_STRING(MB_RegistriHoldingLetti[261]),';');
ADDSTRING(ADR(tempRaw), ADR(temp), tempRawLen);
temp:=CONCAT(INT_TO_STRING(MB_RegistriHoldingLetti[263]),';');
ADDSTRING(ADR(tempRaw), ADR(temp), tempRawLen);
temp:=CONCAT(INT_TO_STRING(MB_RegistriHoldingLetti[264]),';');
ADDSTRING(ADR(tempRaw), ADR(temp), tempRawLen);
temp:=CONCAT(INT_TO_STRING(MB_RegistriHoldingLetti[265]),';');
ADDSTRING(ADR(tempRaw), ADR(temp), tempRawLen);
temp:=CONCAT(INT_TO_STRING(MB_RegistriHoldingLetti[266]),';');
ADDSTRING(ADR(tempRaw), ADR(temp), tempRawLen);
temp:=CONCAT(INT_TO_STRING(MB_RegistriHoldingLetti[267]),';');
ADDSTRING(ADR(tempRaw), ADR(temp), tempRawLen);
temp:=CONCAT(INT_TO_STRING(MB_RegistriHoldingLetti[268]),';');
ADDSTRING(ADR(tempRaw), ADR(temp), tempRawLen);
temp:=CONCAT(INT_TO_STRING(MB_RegistriHoldingLetti[269]),';');
ADDSTRING(ADR(tempRaw), ADR(temp), tempRawLen);
temp:=(INT_TO_STRING(MB_RegistriHoldingLetti[270]));
ADDSTRING(ADR(tempRaw), ADR(temp), tempRawLen);


ADDSTRING(ADR(Logger.TData), ADR(tempRaw), Logger.TLen);
END_ACTION
ACTION CheckAlarm:
(**** GEstione Log ad Evento *****)


	AllarmeCompressore_MB(IN:=MB_RegistriHoldingLetti[1].6 );

	IF AllarmeCompressore_MB.EVH THEN
		LogEv(EL_Alarm,EO_COMPINGRR,ID,1,CONCAT ('AllarmeAttivo_n.', INT_TO_STRING(MB_RegistriHoldingLetti[255])));
	END_IF

	IF AllarmeCompressore_MB.EVL THEN
		LogEv(EL_Log,EO_COMPINGRR,ID,2,CONCAT ('AllarmeRientrato_n.', INT_TO_STRING(MB_RegistriHoldingLetti[255])));
	END_IF
END_ACTION
ACTION Stm:
CASE state OF
	0:	(* Refresh time manager *)
		ReadTmr(IN:=NOT ReadTmr.Q);
		(*A tempo interrogo il nodo sempre che non ci sia qualcuno che lo sta interrogando in quel momento *)

		IF (ReadTmr.Q AND NodoDaInterrogareCompressoreVecchio=Address ) OR Refresh_Now AND NOT InibiscoModbusCompressoreVecchio THEN
			state := 10;
			ReadTmr.PT := T#100ms;  (* moreno *)
			Refresh_Now := FALSE;
			InibiscoModbusCompressoreVecchio := TRUE;
		END_IF

	(**** Leggo le Analogiche a Disposzione  ****)

	10:	(* richiedo lettura Holding Registere   *)

		Modbus.MB_Query.SlaveAddress := Address;
		Modbus.MB_Query.FunctionCode := 3;
		IndirizzoStart:=1;
		ModBus.MB_Query.Read_StartAddress :=IndirizzoStart - 1 ;
		ModBus.MB_Query.Read_Quantity := 2;
		ModBus.MB_Start := TRUE;
		state := 20;

	20:	(* Risposta all'interrogazione *)
		IF NOT ModBus.MB_Start   THEN
			VerificaFuctionCode:=ModBus.MB_Resp.FunctionCode;
			VerificaNodoLetto:=ModBus.MB_Resp.SlaveAddress;

			IF ModBus.MB_MASTER.MB_Error<>0 THEN
				state := 300;
			ELSE
				FOR x:=0 TO ModBus.MB_Query.Read_Quantity DO
					MB_RegistriHoldingLetti[x+IndirizzoStart] := ModBus.MB_Resp.Data[x];   	(* Vedi tabella *)
				END_FOR

					StatusControl[0]:= MB_RegistriHoldingLetti[IndirizzoStart].0;   	(* Vedi tabella *)
					StatusControl[1]:= MB_RegistriHoldingLetti[IndirizzoStart].1;   	(* Vedi tabella *)
					StatusControl[2]:= MB_RegistriHoldingLetti[IndirizzoStart].2;   	(* Vedi tabella *)
					StatusControl[3]:= MB_RegistriHoldingLetti[IndirizzoStart].3;   	(* Vedi tabella *)
					StatusControl[4]:= MB_RegistriHoldingLetti[IndirizzoStart].4;   	(* Vedi tabella *)
					StatusControl[5]:= MB_RegistriHoldingLetti[IndirizzoStart].5;   	(* Vedi tabella *)
					StatusControl[6]:= MB_RegistriHoldingLetti[IndirizzoStart].6;   	(* Vedi tabella *)
					StatusControl[7]:= MB_RegistriHoldingLetti[IndirizzoStart].7;   	(* Vedi tabella *)
					StatusControl[8]:= MB_RegistriHoldingLetti[IndirizzoStart].8;   	(* Vedi tabella *)
					StatusControl[9]:= MB_RegistriHoldingLetti[IndirizzoStart].9;   	(* Vedi tabella *)
					StatusControl[10]:= MB_RegistriHoldingLetti[IndirizzoStart].10;   	(* Vedi tabella *)
					StatusControl[11]:= MB_RegistriHoldingLetti[IndirizzoStart].11;   	(* Vedi tabella *)
					StatusControl[12]:= MB_RegistriHoldingLetti[IndirizzoStart].12;   	(* Vedi tabella *)
					StatusControl[13]:= MB_RegistriHoldingLetti[IndirizzoStart].13;   	(* Vedi tabella *)
					StatusControl[14]:= MB_RegistriHoldingLetti[IndirizzoStart].14;   	(* Vedi tabella *)
					StatusControl[15]:= MB_RegistriHoldingLetti[IndirizzoStart].15;   	(* Vedi tabella *)






				IndirizzoStart:=3;
				ModBus.MB_Query.Read_StartAddress :=IndirizzoStart-1; 	(* richiedo lettura altri Parametri *)
				ModBus.MB_Query.Read_Quantity := 19;
				ModBus.MB_Start := TRUE;

				state := 30;
			END_IF
		END_IF

	30: (* Rispota Altri paramenti *)
		IF NOT ModBus.MB_Start  THEN

			IF ModBus.MB_MASTER.MB_Error<>0 THEN
				state := 300;
			ELSE

				FOR x:=0 TO ModBus.MB_Query.Read_Quantity DO
					MB_RegistriHoldingLetti[x+IndirizzoStart] := ModBus.MB_Resp.Data[x];   	(* Vedi tabella *)
				END_FOR

				IndirizzoStart:=20;
				ModBus.MB_Query.Read_StartAddress :=IndirizzoStart-1; 	(* richiedo lettura altri Parametri *)
				ModBus.MB_Query.Read_Quantity := 1;
				ModBus.MB_Start := TRUE;

				state := 40;
			END_IF
		END_IF

	40: (* Rispota Altri paramenti *)
		IF NOT ModBus.MB_Start  THEN

			IF ModBus.MB_MASTER.MB_Error<>0 THEN
				state := 300;
			ELSE

				FOR x:=0 TO ModBus.MB_Query.Read_Quantity DO
					MB_RegistriHoldingLetti[x+IndirizzoStart] := ModBus.MB_Resp.Data[x];   	(* Vedi tabella *)
				END_FOR

				IndirizzoStart:=64;
				ModBus.MB_Query.Read_StartAddress :=IndirizzoStart-1; 	(* richiedo lettura altri Parametri *)
				ModBus.MB_Query.Read_Quantity := 4;
				ModBus.MB_Start := TRUE;

				state := 45;
			END_IF
		END_IF

	45: (* Rispota Altri paramenti *)
		IF NOT ModBus.MB_Start  THEN

			IF ModBus.MB_MASTER.MB_Error<>0 THEN
				state := 300;
			ELSE
				FOR x:=0 TO ModBus.MB_Query.Read_Quantity DO
					MB_RegistriHoldingLetti[x+IndirizzoStart] := ModBus.MB_Resp.Data[x];   	(* Vedi tabella *)
				END_FOR

				IndirizzoStart:=96;
				ModBus.MB_Query.Read_StartAddress :=IndirizzoStart-1; 	(* richiedo lettura altri Parametri *)
				ModBus.MB_Query.Read_Quantity := 8;
				ModBus.MB_Start := TRUE;

				state := 50;
			END_IF
		END_IF


	50: (* Rispota Altri paramenti *)
		IF NOT ModBus.MB_Start  THEN

			IF ModBus.MB_MASTER.MB_Error<>0 THEN
				state := 300;
			ELSE
				FOR x:=0 TO ModBus.MB_Query.Read_Quantity DO
					MB_RegistriHoldingLetti[x+IndirizzoStart] := ModBus.MB_Resp.Data[x];   	(* Vedi tabella *)
				END_FOR

				IndirizzoStart:=112;
				ModBus.MB_Query.Read_StartAddress :=IndirizzoStart-1; 	(* richiedo lettura altri Parametri *)
				ModBus.MB_Query.Read_Quantity := 10;
				ModBus.MB_Start := TRUE;


				state := 51;
			END_IF
		END_IF


	51: (* Rispota Altri paramenti *)
		IF NOT ModBus.MB_Start  THEN

			IF ModBus.MB_MASTER.MB_Error<>0 THEN
				state := 300;
			ELSE
				FOR x:=0 TO ModBus.MB_Query.Read_Quantity DO
					MB_RegistriHoldingLetti[x+IndirizzoStart] := ModBus.MB_Resp.Data[x];   	(* Vedi tabella *)
				END_FOR

				IndirizzoStart:=256;
				ModBus.MB_Query.Read_StartAddress :=IndirizzoStart-1; 	(* richiedo lettura altri Parametri *)
				ModBus.MB_Query.Read_Quantity := 14;
				ModBus.MB_Start := TRUE;


				state := 55;
			END_IF
		END_IF


	55: (* Rispota Altri paramenti *)
		IF NOT ModBus.MB_Start  THEN

			IF ModBus.MB_MASTER.MB_Error<>0 THEN
				state := 300;
			ELSE
				FOR x:=0 TO ModBus.MB_Query.Read_Quantity DO
					MB_RegistriHoldingLetti[x+IndirizzoStart] := ModBus.MB_Resp.Data[x];   	(* Vedi tabella *)
				END_FOR

				IndirizzoStart:=122;
				ModBus.MB_Query.Read_StartAddress :=IndirizzoStart-1; 	(* richiedo lettura altri Parametri *)
				ModBus.MB_Query.Read_Quantity := 10;
				ModBus.MB_Start := TRUE;

				state := 56;
			END_IF
		END_IF

	56: (* Rispota Altri paramenti *)
		IF NOT ModBus.MB_Start  THEN

			IF ModBus.MB_MASTER.MB_Error<>0 THEN
				state := 300;
			ELSE
				FOR x:=0 TO ModBus.MB_Query.Read_Quantity DO
					MB_RegistriHoldingLetti[x+IndirizzoStart] := ModBus.MB_Resp.Data[x];   	(* Vedi tabella *)
				END_FOR

				IndirizzoStart:=132;
				ModBus.MB_Query.Read_StartAddress :=IndirizzoStart-1; 	(* richiedo lettura altri Parametri *)
				ModBus.MB_Query.Read_Quantity := 10;
				ModBus.MB_Start := TRUE;

				state := 57;
			END_IF
		END_IF

	57: (* Rispota Altri paramenti *)
		IF NOT ModBus.MB_Start  THEN

			IF ModBus.MB_MASTER.MB_Error<>0 THEN
				state := 300;
			ELSE
				FOR x:=0 TO ModBus.MB_Query.Read_Quantity DO
					MB_RegistriHoldingLetti[x+IndirizzoStart] := ModBus.MB_Resp.Data[x];   	(* Vedi tabella *)
				END_FOR

				IndirizzoStart:=142;
				ModBus.MB_Query.Read_StartAddress :=IndirizzoStart-1; 	(* richiedo lettura altri Parametri *)
				ModBus.MB_Query.Read_Quantity := 10;
				ModBus.MB_Start := TRUE;

				state := 58;
			END_IF
		END_IF

	58: (* Rispota Altri paramenti *)
		IF NOT ModBus.MB_Start  THEN

			IF ModBus.MB_MASTER.MB_Error<>0 THEN
				state := 300;
			ELSE
				FOR x:=0 TO ModBus.MB_Query.Read_Quantity DO
					MB_RegistriHoldingLetti[x+IndirizzoStart] := ModBus.MB_Resp.Data[x];   	(* Vedi tabella *)
				END_FOR

				IndirizzoStart:=250;
				ModBus.MB_Query.Read_StartAddress :=IndirizzoStart-1; 	(* richiedo lettura altri Parametri *)
				ModBus.MB_Query.Read_Quantity := 6;
				ModBus.MB_Start := TRUE;

				state := 60;
			END_IF
		END_IF




	60: (* Rispota Altri paramenti *)
		IF NOT ModBus.MB_Start  THEN

			IF ModBus.MB_MASTER.MB_Error<>0 THEN
				state := 300;
			ELSE
				FOR x:=0 TO ModBus.MB_Query.Read_Quantity DO
					MB_RegistriHoldingLetti[x+IndirizzoStart] := ModBus.MB_Resp.Data[x];   	(* Vedi tabella *)
				END_FOR

				state :=290;
			END_IF
		END_IF


		290:    (* Scrittura BOOL - COIL o WORD *)
		IF NOT ModBus.MB_Start THEN
			IF ModBus.MB_MASTER.MB_Error<>0 THEN (*OR ModBus.MB_MASTER.MB_Error<>0 THEN*)
				state := 300;
			ELSE
				IF ScriviDato THEN
					IF ScriviCoil THEN
						Modbus.MB_Query.FunctionCode := 5;
					ELSE
						Modbus.MB_Query.FunctionCode := 6;
					END_IF
					Modbus.MB_Query.SlaveAddress := Address;
					ModBus.MB_Query.Write_StartAddress := IndirizzoDaScrivere-1;
					ModBus.MB_Query.Write_Quantity :=1;

					IF Stop THEN
								 DatoDaScrivere:=MB_RegistriHoldingLetti[IndirizzoDaScrivere];
	  							 DatoDaScrivere.0:=TRUE;
  							        DatoDaScrivere.1:=FALSE;
					END_IF
					IF start THEN
								 DatoDaScrivere:=MB_RegistriHoldingLetti[IndirizzoDaScrivere];
	  							 DatoDaScrivere.0:=TRUE;
  							        DatoDaScrivere.1:=TRUE;
					END_IF

					ModBus.MB_Query.Write_Data[0] := DatoDaScrivere;


					ModBus.MB_Start := TRUE;
						IF ScriviCoil THEN
							IF 	MB_BitStato[IndirizzoDaScrivere]=WORD_TO_BOOL(DatoDaScrivere-1) THEN
								ScriviDato:=FALSE;
							END_IF
						ELSE
							IF 	MB_RegistriHoldingLetti[IndirizzoDaScrivere]=DatoDaScrivere THEN
								ScriviDato:=FALSE;
							END_IF
						END_IF
					state := 295;
				ELSE
					state := 295;
				END_IF
			END_IF
		END_IF




		295:
		IF NOT ModBus.MB_Start THEN
			IF ModBus.MB_MASTER.MB_Error<>0 THEN (*OR ModBus.MB_MASTER.MB_Error<>0 THEN*)
				state := 300;
			ELSE
				IF fModbusAlr THEN fModbusAlr := FALSE; END_IF
				NodoDaInterrogareCompressoreVecchio:=Address+1;
				InibiscoModbusCompressoreVecchio:=FALSE;
				retryErr := 0;
				retry := 0;
				state := 0;
					IF fModbusAlr=FALSE AND ErroreComuModBus=TRUE THEN
						LogEv(EL_Log,EO_COMPINGRR,ID,62,'ComunicazioneModBus_OK');
						ErroreComuModBus := FALSE;
				(*	WarningCtr := SEL(WarningCtr=0, WarningCtr-1, 0); *)
					END_IF


			END_IF
		END_IF



	(**** CHECK MODBUS ERROR ****)
	300: 	(* Release MODBUS *)
			InibiscoModbusCompressoreVecchio:=FALSE;
			(* Retries *)
			retry:=retry+1;
			IF retry>3 THEN
				retry:=0;

				(* Verify if slave is dead *)
				IF retryErr < retryErrMaX THEN
					retryErr := retryErr + 1;
				ELSE
					fModbusAlr := TRUE;
					(* Verify ModBus error	*)

					IF fModbusAlr AND ErroreComuModBus=FALSE THEN
						LogEv(EL_Alarm,EO_COMPINGRR,ID,61,CONCAT('ErroreModbus_',INT_TO_STRING(ModBus.MB_MASTER.MB_Error)));
						ErroreComuModBus := TRUE;
					END_IF
				END_IF

				END_IF
			Refresh_Now := FALSE;
			NodoDaInterrogareCompressoreVecchio:=Address+1;
			state:=0;
END_CASE




(* Controllo Time Out Ciclo ModBus *)

TimeOutModBus(In:=state<>0,PT:=t#30s);
IF TimeOutModBus.Q THEN
	State:=0;
	Refresh_Now:=TRUE;  (* Rilancio la lettura del nodo *)
	IF MODBUS.MB_Lock=TRUE THEN MODBUS.MB_Lock:=FALSE;END_IF
	IF InibiscoModbusCompressoreVecchio=TRUE THEN InibiscoModbusCompressoreVecchio:=FALSE;END_IF
	NodoDaInterrogareCompressoreVecchio:=Address+1;

END_IF
END_ACTION

(* POU Plant_Objects/obj_MisPortata_ETH, ST *)
FUNCTION_BLOCK obj_MisPortata_ETH
(* === MODBUS-TCP PROTOCOL INTERFACE ===
   v1.0[10/06/15] - Create
*)
VAR CONSTANT
	VARS_Max	: BYTE := 32;
END_VAR
VAR_INPUT
	(* Settings *)
	ID			: BYTE;
	IP			: STRING;


(*
	(* Variables management *)
	VARS_En		: BOOL;
	VARS		: ARRAY [0..VARS_Max] OF typ_MODBUS_VAR;
	VARS_Check	: BOOL;
	VARS_Alarm	: BOOL;
	(* Variables allocation *)
	VAR_Pointer : POINTER TO ARRAY[0..99] OF WORD;
	VAR_Cfg		: POINTER TO typ_MODBUS_VAR;    *)
	startCom: BOOL;
END_VAR
VAR_OUTPUT
	(* Status *)
	Status_Log	: BYTE;
	Status_Vis	: DWORD;
END_VAR
VAR
	sta         : BYTE :=0;
	i			: BYTE;
	j			: BYTE;
	Alarm		: FLT_EVENT;

	VarTmr		: TON := (PT:=T#1s);
	VarSta		: BYTE; (* Status *)
	VarCnt		: BYTE; (* Scan counter *)
	VarRetry	: BYTE;
	VarAlarm	: BYTE; (* Last variable with errors *)


	state : INT;
	ReadTmr		:	TON := (PT:=T#5s);
	retry		:	BYTE;
	retryErr	:	BYTE;
	retryErrMax	:	BYTE := 2;

	ErroreComuModBus: BOOL;
	fModbusAlr:BOOL;

	MB_RegistriHoldingLetti: ARRAY [0..300] OF INT;

	x: INT;

	(* da diego per gestione stato stringa > 255*)
	temp :STRING(255);
	tempRaw		: ARRAY [0..MAX_SEND_TCP_CLIENT] OF BYTE;
	tempRawLen :DINT;
	longString:STRING(300);




	TimeOutModBus: TON;
	ErroreTimeOut: BOOL;


	Parametro16:DWORD;
	Parametro18:DWORD;
	Parametro32:DWORD;
	Parametro33:DWORD;
	Parametro64:DWORD;
	Parametro128:DWORD;

	PressioneCalcolata: REAL;
	IntPressioneCalcolata: INT;



END_VAR

VAR_IN_OUT
	(* Interface *)
	MODBUS			: obj_MODBUS_TCP;
END_VAR
CASE state OF
	0:	(* Refresh time manager *)
		(*ReadTmr(IN:=NOT ReadTmr.Q,pt:=t#1s);          ReadTmr.Q *)
		(*	MODBUS.MB_Start:=FALSE; *)

		(*A tempo interrogo il nodo sempre che non ci sia qualcuno che lo sta interrogando in quel momento *)
		IF  startCom   THEN
			state := 10;
		END_IF

			TimeOutModBus(In:=FALSE);


	(**** Leggo le Analogiche a Disposzione  ****)

	10:	(* richiedo lettura Holding Registere   *)

			MODBUS.ID := ID;
			MODBUS.IP := IP;
			MODBUS.MB_MASTER.bFUNCTION_CODE:=3;
			MODBUS.MB_MASTER.wREAD_ADDRESS:=130;
			MODBUS.MB_MASTER.wREAD_QUANTITY:=16;
			MODBUS.MB_Start:=TRUE;
			state := 20;


	20:	(* Risposta all'interrogazione *)
		IF NOT MODBUS.MB_Start  THEN
			IF MODBUS.MB_MASTER.wERROR<>MB_NO_ERROR THEN
				state:=300;
			ELSE


				FOR x:=0 TO MODBUS.MB_MASTER.wREAD_QUANTITY DO
					MB_RegistriHoldingLetti[x+MODBUS.MB_MASTER.wREAD_ADDRESS] := MODBUS.MB_READBUF[x];
				END_FOR


				Parametro16:=MODBUS.MB_READBUF[1]*65535+MODBUS.MB_READBUF[0];
				Parametro18:=MODBUS.MB_READBUF[5]*65535+MODBUS.MB_READBUF[4];



				MODBUS.MB_MASTER.wREAD_ADDRESS:=180;
				MODBUS.MB_MASTER.wREAD_QUANTITY:=4;
				MODBUS.MB_Start:=TRUE;
				state := 30;

			END_IF
		END_IF

	30:	(* Risposta all'interrogazione *)
		IF NOT MODBUS.MB_Start  THEN
			IF MODBUS.MB_MASTER.wERROR<>MB_NO_ERROR THEN
				state:=300;
			ELSE


				FOR x:=0 TO MODBUS.MB_MASTER.wREAD_QUANTITY DO
					MB_RegistriHoldingLetti[x+MODBUS.MB_MASTER.wREAD_ADDRESS] := MODBUS.MB_READBUF[x];
				END_FOR

				Parametro32:=MODBUS.MB_READBUF[1]*65535+MODBUS.MB_READBUF[0];
				Parametro33:=MODBUS.MB_READBUF[3]*65535+MODBUS.MB_READBUF[2];



				MODBUS.MB_MASTER.wREAD_ADDRESS:=230;
				MODBUS.MB_MASTER.wREAD_QUANTITY:=4;
				MODBUS.MB_Start:=TRUE;
				state := 40;

			END_IF
		END_IF

	40:	(* Risposta all'interrogazione *)
		IF NOT MODBUS.MB_Start  THEN
			IF MODBUS.MB_MASTER.wERROR<>MB_NO_ERROR THEN
				state:=300;
			ELSE


				FOR x:=0 TO MODBUS.MB_MASTER.wREAD_QUANTITY DO
					MB_RegistriHoldingLetti[x+MODBUS.MB_MASTER.wREAD_ADDRESS] := MODBUS.MB_READBUF[x];
				END_FOR

				Parametro64:=MODBUS.MB_READBUF[1]*65535+MODBUS.MB_READBUF[0];



				MODBUS.MB_MASTER.wREAD_ADDRESS:=275;
				MODBUS.MB_MASTER.wREAD_QUANTITY:=12;
				MODBUS.MB_Start:=TRUE;
				state := 50;

			END_IF
		END_IF


	50:	(* Risposta all'interrogazione *)
		IF NOT MODBUS.MB_Start  THEN
			IF MODBUS.MB_MASTER.wERROR<>MB_NO_ERROR THEN
				state:=300;
			ELSE


				FOR x:=0 TO MODBUS.MB_MASTER.wREAD_QUANTITY DO
					MB_RegistriHoldingLetti[x+MODBUS.MB_MASTER.wREAD_ADDRESS] := MODBUS.MB_READBUF[x];
				END_FOR

				Parametro128:=MODBUS.MB_READBUF[1]*65535+MODBUS.MB_READBUF[0];



				MODBUS.MB_MASTER.wREAD_ADDRESS:=300;
				MODBUS.MB_MASTER .wREAD_QUANTITY:=2;
				MODBUS.MB_Start:=TRUE;
				state := 60;

			END_IF
		END_IF


	60:	(* Risposta all'interrogazione *)
		IF NOT MODBUS.MB_Start  THEN
			IF MODBUS.MB_MASTER.wERROR<>MB_NO_ERROR THEN
				state:=300;
			ELSE

				FOR x:=0 TO MODBUS.MB_MASTER.wREAD_QUANTITY DO
					MB_RegistriHoldingLetti[x+MODBUS.MB_MASTER.wREAD_ADDRESS] := MODBUS.MB_READBUF[x];
				END_FOR

				state := 295;

			END_IF
		END_IF


		295:
				retryErr := 0;
				retry := 0;
				state := 0;
					IF fModbusAlr=FALSE AND ErroreComuModBus=TRUE THEN
						LogEv(EL_Log,EO_MODBUS_TCP,ID,2,'Comunicazione_ristabilita');
						ErroreComuModBus := FALSE;
				(*	WarningCtr := SEL(WarningCtr=0, WarningCtr-1, 0); *)
					END_IF



	(**** CHECK MODBUS ERROR ****)
	300: 	(* Release MODBUS *)


			retry:=retry+1;
			IF retry>3 THEN
				retry:=0;

				(* Verify if slave is dead *)
				IF retryErr < retryErrMaX THEN
					retryErr := retryErr + 1;
				ELSE
					fModbusAlr := TRUE;
					(* Verify ModBus error	*)

					IF fModbusAlr AND ErroreComuModBus=FALSE THEN
						LogEv(SEL(MODBUS.MB_MASTER.wERROR>0,EL_Wrn,EL_Alarm),EO_MODBUS_TCP,ID,1,WORD_TO_STRING(MODBUS.MB_MASTER.wERROR));
						ErroreComuModBus := TRUE;
					END_IF
				END_IF

			END_IF
			state:=0;
			MODBUS.MB_MASTER.xCONNECT:=FALSE;

END_CASE


(* Controllo Time Out Ciclo ModBus *)

TimeOutModBus(In:=(state<>0 AND  state<>300) ,PT:=t#1s500ms);
IF TimeOutModBus.Q  THEN
	State:=300;
END_IF


(* Log/visu status *)
   IF Alarm.IN   THEN Status_Log:=2; Status_Vis:=COLOR_RED;
	ELSIF ErroreComuModBus  THEN
		Status_Log:=1; Status_Vis:=COLOR_YELLOW;
  	ELSE
		Status_Log:=0; Status_Vis:=COLOR_GREEN;
END_IF
END_FUNCTION_BLOCK
ACTION AddLogData:
Logger.s1:=INSERT('&FTP=',BYTE_TO_STRING(ID),5);
IF ID<10 THEN Logger.s1:=INSERT(Logger.s1,'0',5); END_IF

FOR tempRawLen:=0 TO MAX_SEND_TCP_CLIENT DO
                tempRaw[tempRawLen]:=0;
END_FOR

tempRawLen:=0;


temp:=Logger.s1;
ADDSTRING(ADR(tempRaw), ADR(temp), tempRawLen);

temp:=CONCAT(WORD_TO_STRING(Status_Log),';');
ADDSTRING(ADR(tempRaw), ADR(temp), tempRawLen);
temp:=CONCAT(DWORD_TO_STRING(Parametro16),';');
ADDSTRING(ADR(tempRaw), ADR(temp), tempRawLen);

(* calcolo per passsare la pressione partendo dal psi *)
PressioneCalcolata:=DWORD_TO_REAL(parametro33)*0.068949;
IntPressioneCalcolata:=REAL_TO_INT(PressioneCalcolata*10);

temp:=CONCAT(DWORD_TO_STRING(IntPressioneCalcolata),';');
ADDSTRING(ADR(tempRaw), ADR(temp), tempRawLen);
temp:=CONCAT(DWORD_TO_STRING(Parametro64),';');
ADDSTRING(ADR(tempRaw), ADR(temp), tempRawLen);
temp:=CONCAT(DWORD_TO_STRING(Parametro128),';');

ADDSTRING(ADR(Logger.TData), ADR(tempRaw), Logger.TLen);
END_ACTION

(* POU Plant_Objects/obj_MODBUS_TCP, ST *)
FUNCTION_BLOCK obj_MODBUS_TCP
(* === MODBUS-TCP PROTOCOL INTERFACE ===
   v1.0[10/06/15] - Create
*)
VAR CONSTANT
	VARS_Max	: BYTE := 32;
END_VAR
VAR_INPUT

	(* Settings *)
	ID			: BYTE;
	IP			: STRING;
	PORT		: WORD:=502;
	(* Interface *)
	MB_MASTER	: ETHERNET_MODBUSMASTER_TCP;
	MB_READBUF	: ARRAY [0..128] OF WORD;
	MB_WRITEBUF : ARRAY [0..128] OF WORD;
	MB_Start	: BOOL;
	MB_Lock		: BOOL;
	(* Variables management *)
	VARS_En		: BOOL;
	VARS		: ARRAY [0..VARS_Max] OF typ_MODBUS_VAR;
	VARS_Check	: BOOL;
	VARS_Alarm	: BOOL;
	(* Variables allocation *)
	VAR_Pointer : POINTER TO ARRAY[0..99] OF WORD;
	VAR_Cfg		: POINTER TO typ_MODBUS_VAR;
END_VAR
VAR_OUTPUT
	(* Status *)
	Status_Log	: BYTE;
	Status_Vis	: DWORD;
END_VAR
VAR
	sta         : BYTE :=0;
	i			: BYTE;
	j			: BYTE;
	Alarm		: FLT_EVENT;

	VarTmr		: TON := (PT:=T#1s);
	VarSta		: BYTE; (* Status *)
	VarCnt		: BYTE; (* Scan counter *)
	VarRetry	: BYTE;
	VarAlarm	: BYTE; (* Last variable with errors *)
END_VAR
MB_MASTER( strIP_ADDRESS:=IP, wPORT:=PORT, tTIME_OUT:=T#750MS, (*xCONNECT:=TRUE,*)
		   ptREAD_DATA:=ADR(MB_READBUF), ptSEND_DATA:=ADR(MB_WRITEBUF), xSEND:=MB_Start );

IF sta=0 THEN
	MB_MASTER.xCONNECT:=TRUE;
	sta:=1;
END_IF

(* Process variable management *)
IF VARS_En THEN VARS_Process(); END_IF
(*
(* Check status *)
Alarm(IN:=(MB_MASTER.wERROR<>0));
IF Alarm.EVH THEN
	LogEv(SEL(MB_MASTER.wERROR>0,EL_Wrn,EL_Alarm),EO_MODBUS_TCP,ID,1,WORD_TO_STRING(MB_MASTER.wERROR));
END_IF
IF Alarm.EVL THEN
	LogEv(EL_Log,EO_MODBUS_TCP,ID,2,'');
END_IF
*)
(* Log/visu status *)
   IF Alarm.IN   THEN Status_Log:=2; Status_Vis:=COLOR_RED;
ELSIF Vars_Alarm THEN Status_Log:=1; Status_Vis:=COLOR_YELLOW;
  				 ELSE Status_Log:=0; Status_Vis:=COLOR_GREEN;
END_IF
END_FUNCTION_BLOCK
ACTION VAR_Search:
(* Search VAR with specific pointer if not found return first free VAR
	[Last VAR is not active... used as safe area...] 
*)
j:=VARS_Max;
FOR i := 0 TO VARS_Max-1 DO
	IF VARS[i].Variable=0 AND j>i THEN j:=i; END_IF
	IF VARS[i].Variable=VAR_Pointer THEN
		VAR_Cfg:=ADR(VARS[i]);
		RETURN;
	END_IF
END_FOR
VAR_Cfg:=ADR(VARS[j]);
END_ACTION
ACTION VARS_Process:
(* Update var timers *)
VarTmr(IN:=(NOT VarTmr.Q));
IF VarTmr.Q THEN
	FOR i := 0 TO VARS_Max DO
		IF VARS[i].Refresh_Cnt>0 THEN VARS[i].Refresh_Cnt:=VARS[i].Refresh_Cnt-1; END_IF
	END_FOR
	VARS_Check:=TRUE;
END_IF


(* Process status *)
CASE VarSta OF
	0: (* === Init *)
		VarCnt:=0;
		VarSta:=1;

	1: (* === Wait check signal *)
		IF VARS_Check THEN
			VARS_Check:=FALSE;
			VarCnt:=0;
			VarSta:=2;
		END_IF

	2: (* === Check loop *)
		IF NOT (MB_Lock OR MB_Start) THEN
			WHILE VarCnt<=(VARS_Max-1) AND VarSta=2 DO
				(* Check only active vars *)
				IF VARS[VarCnt].Variable<>0 THEN
					(* Check var auto-refresh on timer checks *)
					IF VARS[VarCnt].Refresh_Time>0 AND VARS[VarCnt].Refresh_Cnt=0 THEN
						VARS[VarCnt].Refresh_Cnt:=VARS[VarCnt].Refresh_Time;
						VarSta:=3;
					END_IF
					(* Check refresh for change or request *)
					CASE VARS[VarCnt].FunCode OF
						5,6,15,16: (* Write functions *)
							IF VARS[VarCnt].Variable_Size=1 THEN
								IF VARS[VarCnt].Variable^<>VARS[VarCnt].Variable_Mirror THEN
									VARS[VarCnt].Variable_Mirror:=VARS[VarCnt].Variable^;
									VarSta:=3;
								END_IF
							ELSE
								IF VARS[VarCnt].Variable_Mirror<>0 THEN
									VARS[VarCnt].Variable_Mirror:=0;
									VarSta:=3;
								END_IF
							END_IF
						1,2,3,4: (* Write functions *)
							IF VARS[VarCnt].Variable_Mirror<>0 THEN
								VARS[VarCnt].Variable_Mirror:=0;
								VarSta:=3;
							END_IF
					END_CASE
				END_IF
				(* Process query *)
				IF VarSta=3 THEN
					MB_Lock:=TRUE;
					MB_MASTER.bUNIT_ID:=VARS[VarCnt].SlaveAddress;
					MB_MASTER.bFUNCTION_CODE:=VARS[VarCnt].FunCode;
					CASE VARS[VarCnt].FunCode OF
						16#5,16#6,16#F,16#10:
							MB_MASTER.wREAD_ADDRESS:=0;
							MB_MASTER.wREAD_QUANTITY:=0;
							MB_MASTER.wWRITE_ADDRESS:=VARS[VarCnt].FunAddress;
							MB_MASTER.wWRITE_QUANTITY:=VARS[VarCnt].Variable_Size;
							IF VARS[VarCnt].Variable_Size=200 THEN
								COPY_32SWAP16(VARS[VarCnt].Variable, ADR(MB_WRITEBUF));
							ELSIF VARS[VarCnt].Variable_Size>1 THEN
								MEMCPY(VARS[VarCnt].Variable, ADR(MB_WRITEBUF), 2*VARS[VarCnt].Variable_Size);
							ELSE
								MB_WRITEBUF[0]:=VARS[VarCnt].Variable^;
							END_IF
						16#1,16#2,16#3,16#4:
							MB_MASTER.wREAD_ADDRESS:=VARS[VarCnt].FunAddress;
							IF VARS[VarCnt].Variable_Size=200 THEN MB_MASTER.wREAD_QUANTITY:=2; ELSE
							  MB_MASTER.wREAD_QUANTITY:=VARS[VarCnt].Variable_Size;
							END_IF
							MB_MASTER.wWRITE_ADDRESS:=0;
							MB_MASTER.wWRITE_QUANTITY:=0;
					END_CASE
					VarRetry:=0;
					MB_Start:=TRUE;
				ELSE
					VarCnt:=VarCnt+1;
				END_IF
			END_WHILE
			(* Check loop completed -> no actions *)
			IF VarSta=2 THEN VarSta:=1; END_IF
		END_IF

	3: (* === Wait & process MB response *)
		IF NOT MB_Start THEN
			IF MB_MASTER.wERROR=0 THEN
				CASE VARS[VarCnt].FunCode OF
					1,2,3,4:
						IF VARS[VarCnt].Variable_Size=200 THEN
							COPY_32SWAP16(ADR(MB_READBUF), VARS[VarCnt].Variable);
						ELSIF VARS[VarCnt].Variable_Size>1 THEN
							MEMCPY(ADR(MB_READBUF), VARS[VarCnt].Variable, 2*VARS[VarCnt].Variable_Size);
						ELSE
							VARS[VarCnt].Variable^:=MB_READBUF[0];
						END_IF
				END_CASE
				MB_Lock:=FALSE;
				(* Signal error recovery *)
				IF VARS_Alarm=TRUE AND VarCnt=VarAlarm THEN
					LogEv(EL_Wrn,EO_MODBUS_TCP,ID,5,'');
					VARS_Alarm:=FALSE;
				END_IF
				(* Next var *)
				VarCnt:=VarCnt+1;
				VarSta:=2;
			ELSE
				IF VarRetry<10 THEN
					VarRetry:=VarRetry+1;
					MB_Start:=TRUE;
				ELSE
					MB_Lock:=FALSE;
					(* Signal error *)
					IF VARS_Alarm=FALSE THEN
						LogEv(EL_Wrn,EO_MODBUS_TCP,ID,3,WORD_TO_STRING(MB_MASTER.wERROR));
						VARS_Alarm:=TRUE;
						VarAlarm:=VarCnt-1;
					END_IF
					(* Next var *)
					VarCnt:=VarCnt+1;
					VarSta:=2;
				END_IF
			END_IF
		END_IF

ELSE
	VarSta:=0;
END_CASE
END_ACTION

(* POU Plant_Objects/obj_MisPortata_MB, ST *)
FUNCTION_BLOCK obj_MisPortata_MB
VAR CONSTANT
	TimeOutModBus: TON;
END_VAR
VAR_INPUT
	ID			:	BYTE;
	Address		:	BYTE;

	(* Modbus *)
	Refresh_Now	:	BOOL;			(* Richiesta di lettura stato macchina Immediata  *)
	retryErrMax	:	BYTE := 2;

	OnOff		: 	BOOL;

	IndirizzoDaScrivere: WORD;
	DatoDaScrivere: INT;
	ScriviDato: BOOL;
	ScriviCoil: BOOL;

	fWriteAttivazioneComandi:BOOL;

END_VAR
VAR_IN_OUT
	ModBus		:obj_MODBUS;
END_VAR
VAR_OUTPUT
	Run			:	BOOL;

	Status_Log	:	WORD;
	Status_Vis	:	DWORD;
END_VAR
VAR
	(* da diego per gestione stato stringa > 255*)
	temp :STRING(255);
	tempRaw		: ARRAY [0..MAX_SEND_TCP_CLIENT] OF BYTE;
	tempRawLen :DINT;
	longString:STRING(255);

	(* Timer manage switch on/off delay *)
	Delay		: 	TONOF;
	Warning		:	FLT_TAP := (TAP:=100);
	AllarmeCompressore_MB		:	FLT_TAP;

	state		:	INT;
	retry		:	BYTE;
	retryErr	:	BYTE;
	ReadTmr		:	TON := (PT:=T#5s);
	fModbusAlr:BOOL;

	Ctrl_Run: BOOL;


	VerificaFuctionCode: INT;
	VerificaNodoLetto: INT;
	ErroreComuModBus: BOOL;
	IndiceErrore: BYTE;

(*	MB_BitStato: ARRAY [0..1] OF BOOL;
	MB_RegistriLetti: ARRAY [0..1] OF INT;
	MB_RegistriHoldingLetti: ARRAY [0..255] OF WORD;
	MB_BitStatoCoil: ARRAY [0..1] OF BOOL; *)


	Parametro16:DWORD;
	Parametro17:DWORD;
	Parametro18:DWORD;
	Parametro19:DWORD;
	Parametro20:DWORD;
	Parametro21:DWORD;
	Parametro32:DWORD;
	Parametro33:DWORD;
	Parametro64:DWORD;
	Parametro65:DWORD;
	Parametro128:DWORD;





	AddressRead: BYTE;
	index: BYTE;
	indexErr: BYTE;





	x: INT;

	PressioneCalcolata: REAL;
	IntPressioneCalcolata: INT;
END_VAR
(* Call ModBus state machine *)
Stm();


(* Seganalzione stato Compressore  *)
IF ErroreComuModBus THEN
		Status_Log:=2; Status_Vis:=16#2020F0;
(*	ELSIF Warning OR Warning2 THEN
		Status_Log:=1; Status_Vis:=16#20F0F0; *)
    ELSE
		Status_Log:=0;
		Status_Vis:=16#006000;
END_IF
END_FUNCTION_BLOCK
ACTION AddLogData:
Logger.s1:=INSERT('&FTP=',BYTE_TO_STRING(ID),4);
IF ID<10 THEN Logger.s1:=INSERT(Logger.s1,'0',4); END_IF

FOR tempRawLen:=0 TO MAX_SEND_TCP_CLIENT DO
                tempRaw[tempRawLen]:=0;
END_FOR

tempRawLen:=0;


temp:=Logger.s1;
ADDSTRING(ADR(tempRaw), ADR(temp), tempRawLen);

temp:=CONCAT(WORD_TO_STRING(Status_Log),';');
ADDSTRING(ADR(tempRaw), ADR(temp), tempRawLen);
temp:=CONCAT(DWORD_TO_STRING(Parametro16),';');
ADDSTRING(ADR(tempRaw), ADR(temp), tempRawLen);


(* calcolo per passsare la pressione partendo dal psi *)
PressioneCalcolata:=DWORD_TO_REAL(parametro33)*0.068949;
IntPressioneCalcolata:=REAL_TO_INT(PressioneCalcolata*10);

temp:=CONCAT(DWORD_TO_STRING(IntPressioneCalcolata),';');
ADDSTRING(ADR(tempRaw), ADR(temp), tempRawLen);
temp:=CONCAT(DWORD_TO_STRING(Parametro64),';');
ADDSTRING(ADR(tempRaw), ADR(temp), tempRawLen);
temp:=CONCAT(DWORD_TO_STRING(Parametro128),';');

ADDSTRING(ADR(Logger.TData), ADR(tempRaw), Logger.TLen);
END_ACTION
ACTION Stm:
CASE state OF
	0:	(* Refresh time manager *)
		ReadTmr(IN:=NOT ReadTmr.Q);
		(*A tempo interrogo il nodo sempre che non ci sia qualcuno che lo sta interrogando in quel momento *)

		IF (ReadTmr.Q AND NodoDaInterrogareMisuratoreDiPortata=Address ) OR Refresh_Now AND NOT InibiscoModbusMisuratoreDiPortata THEN
			state := 10;
			ReadTmr.PT := T#500ms;  (* moreno *)
			Refresh_Now := FALSE;
			InibiscoModbusMisuratoreDiPortata := TRUE;
		END_IF

	(**** Leggo le Analogiche a Disposzione  ****)

	10:	(* richiedo lettura Holding Registere   *)

		Modbus.MB_Query.SlaveAddress := Address;
		Modbus.MB_Query.FunctionCode := 3;
		ModBus.MB_Query.Read_StartAddress := 16; (* 41 ; *)
		ModBus.MB_Query.Read_Quantity :=2;
		ModBus.MB_Start := TRUE;
		state := 20;

	20:	(* Risposta all'interrogazione *)
		IF NOT ModBus.MB_Start   THEN
			VerificaFuctionCode:=ModBus.MB_Resp.FunctionCode;
			VerificaNodoLetto:=ModBus.MB_Resp.SlaveAddress;

			IF ModBus.MB_MASTER.MB_Error<>0 THEN
				state := 300;
			ELSE
			(*	FOR x:=0 TO ModBus.MB_Query.Read_Quantity DO
					MB_RegistriHoldingLetti[x+ModBus.MB_Query.Read_StartAddress] := ModBus.MB_Resp.Data[x];   	(* Vedi tabella *)
				END_FOR *)

				Parametro16:=ModBus.MB_Resp.Data[1]*65535+ModBus.MB_Resp.Data[0];


				ModBus.MB_Query.Read_StartAddress :=17; 	(* richiedo lettura altri Parametri *)
				ModBus.MB_Query.Read_Quantity := 2;
				ModBus.MB_Start := TRUE;

				state := 30;
			END_IF
		END_IF

	30: (* Rispota Altri paramenti *)
		IF NOT ModBus.MB_Start  THEN

			IF ModBus.MB_MASTER.MB_Error<>0 THEN
				state := 300;
			ELSE

			(*	FOR x:=0 TO ModBus.MB_Query.Read_Quantity DO
					MB_RegistriHoldingLetti[x+ModBus.MB_Query.Read_StartAddress] := ModBus.MB_Resp.Data[x];   	(* Vedi tabella *)
				END_FOR *)


				Parametro17:=ModBus.MB_Resp.Data[1]*65535+ModBus.MB_Resp.Data[0];


				ModBus.MB_Query.Read_StartAddress :=18; 	(* richiedo lettura altri Parametri *)
				ModBus.MB_Query.Read_Quantity := 2;
				ModBus.MB_Start := TRUE;

				state := 40;
			END_IF
		END_IF


	40: (* Rispota Altri paramenti *)
		IF NOT ModBus.MB_Start  THEN

			IF ModBus.MB_MASTER.MB_Error<>0 THEN
				state := 300;
			ELSE

			(*	FOR x:=0 TO ModBus.MB_Query.Read_Quantity DO
					MB_RegistriHoldingLetti[x+ModBus.MB_Query.Read_StartAddress] := ModBus.MB_Resp.Data[x];   	(* Vedi tabella *)
				END_FOR *)



				Parametro18:=ModBus.MB_Resp.Data[1]*65535+ModBus.MB_Resp.Data[0];


				ModBus.MB_Query.Read_StartAddress :=19; 	(* richiedo lettura altri Parametri *)
				ModBus.MB_Query.Read_Quantity := 2;
				ModBus.MB_Start := TRUE;

				state := 50;
			END_IF
		END_IF

	50: (* Rispota Altri paramenti *)
		IF NOT ModBus.MB_Start  THEN

			IF ModBus.MB_MASTER.MB_Error<>0 THEN
				state := 300;
			ELSE

			(*	FOR x:=0 TO ModBus.MB_Query.Read_Quantity DO
					MB_RegistriHoldingLetti[x+ModBus.MB_Query.Read_StartAddress] := ModBus.MB_Resp.Data[x];   	(* Vedi tabella *)
				END_FOR *)


				Parametro19:=ModBus.MB_Resp.Data[1]*65535+ModBus.MB_Resp.Data[0];


				ModBus.MB_Query.Read_StartAddress :=20; 	(* richiedo lettura altri Parametri *)
				ModBus.MB_Query.Read_Quantity := 2;
				ModBus.MB_Start := TRUE;

				state := 60;
			END_IF
		END_IF

	60: (* Rispota Altri paramenti *)
		IF NOT ModBus.MB_Start  THEN

			IF ModBus.MB_MASTER.MB_Error<>0 THEN
				state := 300;
			ELSE

			(*	FOR x:=0 TO ModBus.MB_Query.Read_Quantity DO
					MB_RegistriHoldingLetti[x+ModBus.MB_Query.Read_StartAddress] := ModBus.MB_Resp.Data[x];   	(* Vedi tabella *)
				END_FOR *)


				Parametro20:=ModBus.MB_Resp.Data[1]*65535+ModBus.MB_Resp.Data[0];


				ModBus.MB_Query.Read_StartAddress :=21; 	(* richiedo lettura altri Parametri *)
				ModBus.MB_Query.Read_Quantity := 2;
				ModBus.MB_Start := TRUE;

				state := 70;
			END_IF
		END_IF

	70: (* Rispota Altri paramenti *)
		IF NOT ModBus.MB_Start  THEN

			IF ModBus.MB_MASTER.MB_Error<>0 THEN
				state := 300;
			ELSE

			(*	FOR x:=0 TO ModBus.MB_Query.Read_Quantity DO
					MB_RegistriHoldingLetti[x+ModBus.MB_Query.Read_StartAddress] := ModBus.MB_Resp.Data[x];   	(* Vedi tabella *)
				END_FOR *)


				Parametro21:=ModBus.MB_Resp.Data[1]*65535+ModBus.MB_Resp.Data[0];


				ModBus.MB_Query.Read_StartAddress :=32; 	(* richiedo lettura altri Parametri *)
				ModBus.MB_Query.Read_Quantity := 2;
				ModBus.MB_Start := TRUE;

				state := 80;
			END_IF
		END_IF

	80: (* Rispota Altri paramenti *)
		IF NOT ModBus.MB_Start  THEN

			IF ModBus.MB_MASTER.MB_Error<>0 THEN
				state := 300;
			ELSE

			(*	FOR x:=0 TO ModBus.MB_Query.Read_Quantity DO
					MB_RegistriHoldingLetti[x+ModBus.MB_Query.Read_StartAddress] := ModBus.MB_Resp.Data[x];   	(* Vedi tabella *)
				END_FOR *)


				Parametro32:=ModBus.MB_Resp.Data[1]*65535+ModBus.MB_Resp.Data[0];


				ModBus.MB_Query.Read_StartAddress :=33; 	(* richiedo lettura altri Parametri *)
				ModBus.MB_Query.Read_Quantity := 2;
				ModBus.MB_Start := TRUE;

				state := 90;
			END_IF
		END_IF

	90: (* Rispota Altri paramenti *)
		IF NOT ModBus.MB_Start  THEN

			IF ModBus.MB_MASTER.MB_Error<>0 THEN
				state := 300;
			ELSE

			(*	FOR x:=0 TO ModBus.MB_Query.Read_Quantity DO
					MB_RegistriHoldingLetti[x+ModBus.MB_Query.Read_StartAddress] := ModBus.MB_Resp.Data[x];   	(* Vedi tabella *)
				END_FOR *)


				Parametro33:=ModBus.MB_Resp.Data[1]*65535+ModBus.MB_Resp.Data[0];


				ModBus.MB_Query.Read_StartAddress :=64; 	(* richiedo lettura altri Parametri *)
				ModBus.MB_Query.Read_Quantity := 2;
				ModBus.MB_Start := TRUE;

				state :=100;
			END_IF
		END_IF

	100: (* Rispota Altri paramenti *)
		IF NOT ModBus.MB_Start  THEN

			IF ModBus.MB_MASTER.MB_Error<>0 THEN
				state := 300;
			ELSE

			(*	FOR x:=0 TO ModBus.MB_Query.Read_Quantity DO
					MB_RegistriHoldingLetti[x+ModBus.MB_Query.Read_StartAddress] := ModBus.MB_Resp.Data[x];   	(* Vedi tabella *)
				END_FOR *)


				Parametro64:=ModBus.MB_Resp.Data[1]*65535+ModBus.MB_Resp.Data[0];


				ModBus.MB_Query.Read_StartAddress :=65; 	(* richiedo lettura altri Parametri *)
				ModBus.MB_Query.Read_Quantity := 2;
				ModBus.MB_Start := TRUE;

				state := 110;
			END_IF
		END_IF

	110: (* Rispota Altri paramenti *)
		IF NOT ModBus.MB_Start  THEN

			IF ModBus.MB_MASTER.MB_Error<>0 THEN
				state := 300;
			ELSE

			(*	FOR x:=0 TO ModBus.MB_Query.Read_Quantity DO
					MB_RegistriHoldingLetti[x+ModBus.MB_Query.Read_StartAddress] := ModBus.MB_Resp.Data[x];   	(* Vedi tabella *)
				END_FOR *)


				Parametro65:=ModBus.MB_Resp.Data[1]*65535+ModBus.MB_Resp.Data[0];


				ModBus.MB_Query.Read_StartAddress :=128; 	(* richiedo lettura altri Parametri *)
				ModBus.MB_Query.Read_Quantity := 2;
				ModBus.MB_Start := TRUE;

				state := 120;
			END_IF
		END_IF

	120: (* Rispota Altri paramenti *)
		IF NOT ModBus.MB_Start  THEN

			IF ModBus.MB_MASTER.MB_Error<>0 THEN
				state := 300;
			ELSE

			(*	FOR x:=0 TO ModBus.MB_Query.Read_Quantity DO
					MB_RegistriHoldingLetti[x+ModBus.MB_Query.Read_StartAddress] := ModBus.MB_Resp.Data[x];   	(* Vedi tabella *)
				END_FOR *)


				Parametro128:=ModBus.MB_Resp.Data[1]*65535+ModBus.MB_Resp.Data[0];


				state :=295;
			END_IF
		END_IF


(*




	290:    (* Scrittura BOOL - COIL o WORD *)
		IF NOT ModBus.MB_Start THEN
			IF ModBus.MB_MASTER.MB_Error<>0 THEN (*OR ModBus.MB_MASTER.MB_Error<>0 THEN*)
				state := 300;
			ELSE
				IF ScriviDato THEN
					IF ScriviCoil THEN
						Modbus.MB_Query.FunctionCode := 5;
					ELSE
						Modbus.MB_Query.FunctionCode := 6;
					END_IF
					Modbus.MB_Query.SlaveAddress := Address;
					ModBus.MB_Query.Write_StartAddress := IndirizzoDaScrivere;
					ModBus.MB_Query.Write_Quantity :=1;
					ModBus.MB_Query.Write_Data[0] := DatoDaScrivere;
					ModBus.MB_Start := TRUE;
						IF ScriviCoil THEN
							IF 	MB_BitStato[IndirizzoDaScrivere]=WORD_TO_BOOL(DatoDaScrivere-1) THEN
								ScriviDato:=FALSE;
							END_IF
						ELSE
							IF 	MB_RegistriLetti[IndirizzoDaScrivere]=DatoDaScrivere THEN
								ScriviDato:=FALSE;
							END_IF
						END_IF
					state := 295;
				ELSE
					state := 295;
				END_IF
			END_IF
		END_IF


*)

		295:
		IF NOT ModBus.MB_Start THEN
			IF ModBus.MB_MASTER.MB_Error<>0 THEN (*OR ModBus.MB_MASTER.MB_Error<>0 THEN*)
				state := 300;
			ELSE
				IF fModbusAlr THEN fModbusAlr := FALSE; END_IF
				NodoDaInterrogareMisuratoreDiPortata:=Address+1;
				InibiscoModbusMisuratoreDiPortata:=FALSE;
				retryErr := 0;
				retry := 0;
				state := 0;
					IF fModbusAlr=FALSE AND ErroreComuModBus=TRUE THEN
						LogEv(EL_Log,EO_FPT,ID,62,'ComunicazioneModBus_OK');
						ErroreComuModBus := FALSE;
				(*	WarningCtr := SEL(WarningCtr=0, WarningCtr-1, 0); *)
					END_IF


			END_IF
		END_IF



	(**** CHECK MODBUS ERROR ****)
	300: 	(* Release MODBUS *)
			InibiscoModbusMisuratoreDiPortata:=FALSE;
			(* Retries *)
			retry:=retry+1;
			IF retry>3 THEN
				retry:=0;

				(* Verify if slave is dead *)
				IF retryErr < retryErrMaX THEN
					retryErr := retryErr + 1;
				ELSE
					fModbusAlr := TRUE;
					(* Verify ModBus error	*)

					IF fModbusAlr AND ErroreComuModBus=FALSE THEN
						LogEv(EL_Alarm,EO_FPT,ID,61,CONCAT('ErroreModbus_',INT_TO_STRING(ModBus.MB_MASTER.MB_Error)));
						ErroreComuModBus := TRUE;
					END_IF
				END_IF

				END_IF
			Refresh_Now := FALSE;
			NodoDaInterrogareMisuratoreDiPortata:=Address+1;
			state:=0;
END_CASE


(* calcolo per passsare la pressione partendo dal psi *)
PressioneCalcolata:=DWORD_TO_REAL(parametro33)*0.06895;
IntPressioneCalcolata:=REAL_TO_INT(PressioneCalcolata*10);



(* Controllo Time Out Ciclo ModBus *)

TimeOutModBus(In:=state<>0,PT:=t#30s);
IF TimeOutModBus.Q THEN
	State:=0;
	Refresh_Now:=TRUE;  (* Rilancio la lettura del nodo *)
	IF MODBUS.MB_Lock=TRUE THEN MODBUS.MB_Lock:=FALSE;END_IF
	IF InibiscoModbusMisuratoreDiPortata=TRUE THEN InibiscoModbusMisuratoreDiPortata:=FALSE;END_IF
	NodoDaInterrogareMisuratoreDiPortata:=Address+1;

END_IF
END_ACTION

(* POU Utils Functions/PLANT_STATUS, ST *)
FUNCTION_BLOCK PLANT_STATUS
VAR_INPUT
	obj_Status		:	WORD;
END_VAR
VAR_OUTPUT
END_VAR
VAR
	PLANT_STATUS	:	WORD;

	Pwm				:	TON := (PT:=T#1s);
END_VAR
CASE plant_Status OF

	0:	(* Plant OK - Everything works well *)
		Pwm(IN:=FALSE);							(* Stop timer if running *)
		LAMP_AL := FALSE;						(* Keep the lamp switched off *)

	1:	(* Plant in warning *)
		Pwm(IN:= NOT(Pwm.Q));

		IF Pwm.Q THEN
			LAMP_AL := NOT LAMP_AL;				(* Toggle output *)
		END_IF

	2:	(* Plant in alarm *)
		Pwm(IN:=FALSE);							(* Stop timer if running *)
		LAMP_AL	:= TRUE;						(* Keep the lamp switched on *)

END_CASE

plant_Status := 0;		(* Reset plant status *)
END_FUNCTION_BLOCK
ACTION UpdateStatus:
IF plant_Status = 2 THEN

	RETURN;					(* If plant already in alarm condition do nothing *)

ELSE

		IF obj_Status <> 0 THEN
			plant_Status := obj_Status;			(* If plant in warning/normal condition and current object in alarm, update plant status *)
		END_IF
END_IF
END_ACTION

(* POU PLC_WDT, ST *)
FUNCTION PLC_WDT: DWORD VAR_INPUT dwEvent: DWORD; dwFilter: DWORD; dwOwner: DWORD; END_VAR
LogEv(EL_AlarmStop,EO_SYS,1,10,'Watchdog');
END_FUNCTION

(* POU Utils Functions/RAWTOHEXSTR, ST *)
FUNCTION RAWTOHEXSTR : STRING(128)
VAR_INPUT
	pData: POINTER TO BYTE;
	DataLen: BYTE;
END_VAR
VAR
	pt: POINTER TO BYTE;
	xl: BYTE;
END_VAR
pt:=ADR(RAWTOHEXSTR);

xl:=2;

WHILE DataLen>0 AND xl<128 DO

	pt^ := (pData^ / 16#10) + 48 + (((pData^ / 16#10)/10)*7);
	pt:=pt+1;
	pt^ := (pData^ AND 16#0F)  + 48 + (((pData^ AND 16#0F)/10)*7);
	pt:=pt+1;

	xl:=xl+2;

	DataLen:=DataLen-1;
	pData:=pData+1;

END_WHILE

pt^:=0;
END_FUNCTION

(* POU Utils/RTC_Update, ST *)
FUNCTION RTC_Update : BOOL
VAR
	T: DT;
	TS: STRING;
	TS2: STRING;
	Hour: BYTE;
	Minute: BYTE;
END_VAR
(* Get RTC time *)
T:=SysRtcGetTime(TRUE);
Sys.Time_CT_DT:=T;
(* Calculate variables *)
TS:=DT_TO_STRING(T);
Sys.Time_LogString:=DELETE(STR:=TS, LEN:=3, POS:=1);
TS2:=MID(STR:=TS, LEN:=4, POS:= 4); Sys.Time_Year 	:=STRING_TO_WORD(TS2);
TS2:=MID(STR:=TS, LEN:=2, POS:= 9); Sys.Time_Month	:=STRING_TO_BYTE(TS2);
TS2:=MID(STR:=TS, LEN:=2, POS:=12); Sys.Time_Day  	:=STRING_TO_BYTE(TS2);
Sys.Time_CT_Day:=(32*(Sys.Time_Month-1)+Sys.Time_Day-1);
TS2:=MID(STR:=TS, LEN:=2, POS:=15); Hour			:=STRING_TO_BYTE(TS2);
TS2:=MID(STR:=TS, LEN:=2, POS:=18); Minute		 	:=STRING_TO_BYTE(TS2);
Sys.Time_CT_Quarter:=Hour*4+(Minute/15);
END_FUNCTION

(* POU Utils Functions/SHIFT_ARRAY, ST *)
FUNCTION SHIFT_ARRAY : BOOL
VAR_INPUT
	pData	:	POINTER TO ARRAY [1..2] OF WORD;
	Size	:	BYTE;
END_VAR
VAR
	pNew	:	POINTER TO WORD;
	i		:	BYTE;
END_VAR
(* Shift right *)
FOR i:=1 TO (Size-1) BY 1 DO

	(*pNew := pData + 1;*)
	pData^[i] := pData^[i+1];
	(*pData := pData + 1;*)

END_FOR
END_FUNCTION

(* Visualisation PLC_VISU
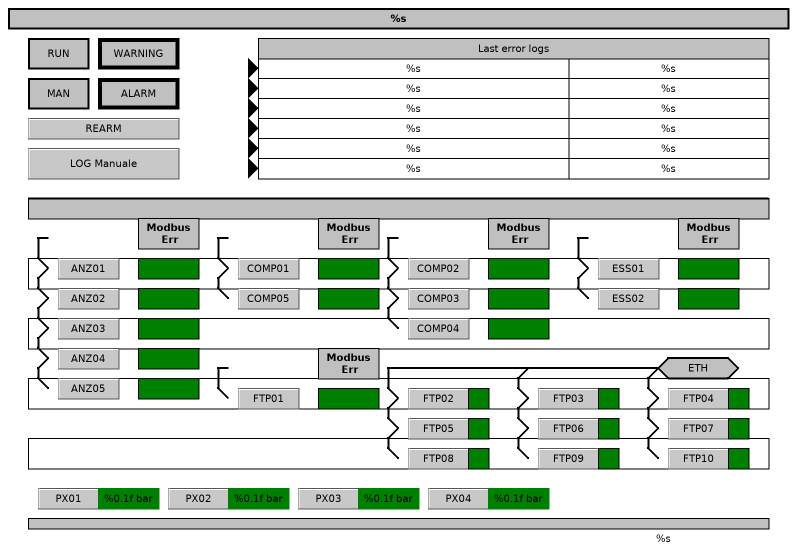
rectangle at (10,0)-(791,21): text "%s"; shows .Plant_NAME
rounded rectangle at (30,30)-(91,61): text "RUN"; alarm colour if NOT Mode_Manual; runs INTERN ASSIGN Mode_Manual:=(FALSE)
rounded rectangle at (30,70)-(91,101): text "MAN"; alarm colour if Mode_Manual; runs INTERN ASSIGN Mode_Manual:=(TRUE)
rectangle at (570,50)-(771,71): text "%s"; shows Sys.LastLogs_Msg[0]
polygon at (250,150)-(260,170): invisible if Sys.LastLogs_Idx<>0
rectangle at (570,70)-(771,91): text "%s"; shows Sys.LastLogs_Msg[1]
polygon at (250,50)-(260,70): invisible if Sys.LastLogs_Idx<>1
rectangle at (570,90)-(771,111): text "%s"; shows Sys.LastLogs_Msg[2]
polygon at (250,70)-(260,90): invisible if Sys.LastLogs_Idx<>2
rectangle at (570,110)-(771,131): text "%s"; shows Sys.LastLogs_Msg[3]
polygon at (250,90)-(260,110): invisible if Sys.LastLogs_Idx<>3
rectangle at (570,130)-(771,151): text "%s"; shows Sys.LastLogs_Msg[4]
polygon at (250,110)-(260,130): invisible if Sys.LastLogs_Idx<>4
rectangle at (570,150)-(771,171): text "%s"; shows Sys.LastLogs_Msg[5]
polygon at (250,130)-(260,150): invisible if Sys.LastLogs_Idx<>5
rectangle at (260,50)-(571,71): text "%s"; shows Sys.LastLogs_Dat[0]
rectangle at (260,70)-(571,91): text "%s"; shows Sys.LastLogs_Dat[1]
rectangle at (260,90)-(571,111): text "%s"; shows Sys.LastLogs_Dat[2]
rectangle at (260,110)-(571,131): text "%s"; shows Sys.LastLogs_Dat[3]
rectangle at (260,130)-(571,151): text "%s"; shows Sys.LastLogs_Dat[4]
rectangle at (260,150)-(571,171): text "%s"; shows Sys.LastLogs_Dat[5]
rectangle at (100,70)-(181,101): text "ALARM"; alarm colour if Sys.Alarm; runs INTERN ASSIGN Mode_Manual:=(FALSE)
rectangle at (100,30)-(181,61): text "WARNING"; alarm colour if Sys.Warning; runs INTERN ASSIGN Mode_Manual:=(TRUE)
button at (30,110)-(181,131): text "REARM"; runs INTERN ASSIGN Sys.Alarm:=(FALSE);INTERN ASSIGN Sys.Warning:=(FALSE)
button at (60,250)-(121,271): text "ANZ01"
rectangle at (260,30)-(771,51): text "Last error logs"
button at (60,280)-(121,301): text "ANZ02"
rectangle at (560,520)-(771,541): text "%s"; shows Sys.Time_LogString
rectangle at (140,210)-(201,241): text "Modbus / Err"
rectangle at (140,280)-(201,301): alarm colour if ANZ_MODBUS_CONNECTOR_INEPRO[2].fTimeout
button at (60,310)-(121,331): text "ANZ03"
rectangle at (140,310)-(201,331): alarm colour if ANZ_MODBUS_CONNECTOR_INEPRO[3].fTimeout
rectangle at (140,250)-(201,271): alarm colour if ANZ_MODBUS_CONNECTOR_INEPRO[1].fTimeout
button at (60,340)-(121,361): text "ANZ04"
rectangle at (140,340)-(201,361): alarm colour if ANZ_MODBUS_CONNECTOR_INEPRO[4].fTimeout
button at (60,370)-(121,391): text "ANZ05"
rectangle at (140,370)-(201,391): alarm colour if ANZ_MODBUS_CONNECTOR_INEPRO[5].fTimeout
button at (240,250)-(301,271): text "COMP01"
button at (240,280)-(301,301): text "COMP05"
rectangle at (320,250)-(381,271): alarm colour if .COMPRESSORE01.ErroreComuModBus
rectangle at (320,280)-(381,301): alarm colour if .COMPRESSORE05.ErroreComuModBus
rectangle at (320,210)-(381,241): text "Modbus / Err"
button at (410,250)-(471,271): text "COMP02"
button at (410,280)-(471,301): text "COMP03"
rectangle at (490,250)-(551,271): alarm colour if .COMPRESSORE02.ErroreComuModBus
rectangle at (490,280)-(551,301): alarm colour if .COMPRESSORE03.ErroreComuModBus
rectangle at (490,210)-(551,241): text "Modbus / Err"
button at (600,250)-(661,271): text "ESS01"
button at (600,280)-(661,301): text "ESS02"
rectangle at (680,250)-(741,271): alarm colour if .COMPRESSORE01.ErroreComuModBus
rectangle at (680,280)-(741,301): alarm colour if .COMPRESSORE05.ErroreComuModBus
rectangle at (680,210)-(741,241): text "Modbus / Err"
button at (240,380)-(301,401): text "FTP01"
rectangle at (320,380)-(381,401): alarm colour if .FTP01.ErroreComuModBus
rectangle at (320,340)-(381,371): text "Modbus / Err"
button at (410,310)-(471,331): text "COMP04"
rectangle at (490,310)-(551,331): alarm colour if .COMPRESSORE04.ErroreComuModBus
button at (40,480)-(101,501): text "PX01"
rectangle at (100,480)-(161,501): text "%0.1f bar"; shows INT_TO_REAL(.PX01.ValoreScalato)/10
button at (170,480)-(231,501): text "PX02"
rectangle at (230,480)-(291,501): text "%0.1f bar"; shows INT_TO_REAL(.PX02.ValoreScalato)/10
button at (300,480)-(361,501): text "PX03"
rectangle at (360,480)-(421,501): text "%0.1f bar"; shows INT_TO_REAL(.PX03.ValoreScalato)/10
button at (430,480)-(491,501): text "PX04"
rectangle at (490,480)-(551,501): text "%0.1f bar"; shows INT_TO_REAL(.PX04.ValoreScalato)/10
button at (30,140)-(181,171): text "LOG Manuale"; taps PLC_PRG.HMI_AggiornaLog
button at (410,380)-(471,401): text "FTP02"
polygon at (660,350)-(740,370): text "ETH"
rectangle at (470,380)-(491,401): alarm colour if .FPT02.ErroreComuModBus
button at (540,380)-(601,401): text "FTP03"
rectangle at (600,380)-(621,401): alarm colour if .FPT03.ErroreComuModBus
button at (670,380)-(731,401): text "FTP04"
rectangle at (730,380)-(751,401): alarm colour if .FPT04.ErroreComuModBus
button at (410,410)-(471,431): text "FTP05"
rectangle at (470,410)-(491,431): alarm colour if .FPT05.ErroreComuModBus
button at (540,410)-(601,431): text "FTP06"
rectangle at (600,410)-(621,431): alarm colour if .FPT06.ErroreComuModBus
button at (670,410)-(731,431): text "FTP07"
rectangle at (730,410)-(751,431): alarm colour if .FPT07.ErroreComuModBus
button at (670,440)-(731,461): text "FTP10"
rectangle at (730,440)-(751,461): alarm colour if .FPT10.ErroreComuModBus
button at (540,440)-(601,461): text "FTP09"
rectangle at (600,440)-(621,461): alarm colour if .FPT09.ErroreComuModBus
button at (410,440)-(471,461): text "FTP08"
rectangle at (470,440)-(491,461): alarm colour if .FPT08.ErroreComuModBus
29 more shapes without text or variables
27 elements of other kinds (tables, trends, ...) not read
*)

(* Visualisation PLC_VISU_raw_data
rectangle at (10,0)-(871,21): text "%s"; shows .Plant_NAME
3 elements of other kinds (tables, trends, ...) not read
*)

(* Visualisation PLC_VISU_raw_data_BIS
rectangle at (10,0)-(791,21): text "%s"; shows .Plant_NAME
3 elements of other kinds (tables, trends, ...) not read
*)

(* Visualisation PLC_VISU_raw_data_tris
rectangle at (10,0)-(791,21): text "%s"; shows .Plant_NAME
2 elements of other kinds (tables, trends, ...) not read
*)

(* Visualisation VIS_SET
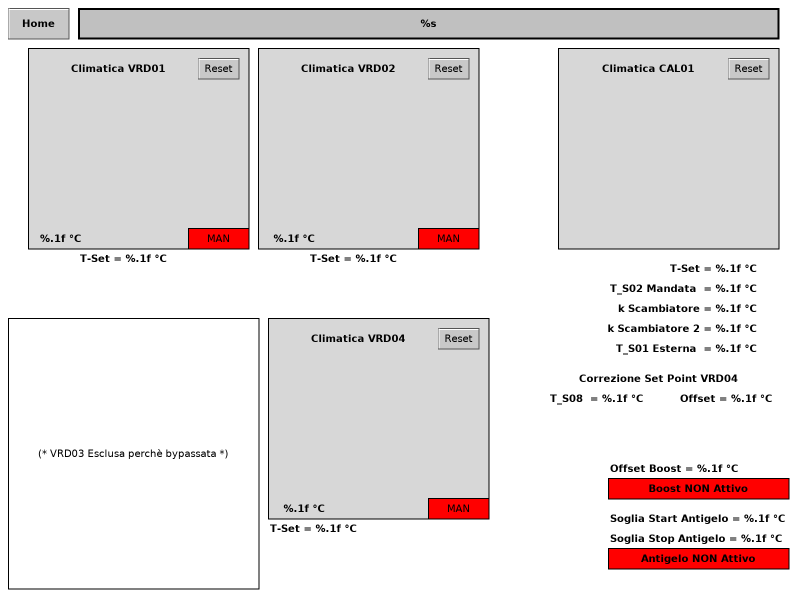
rectangle at (40,60)-(201,81): text "Climatica VRD01"
button at (200,60)-(241,81): text "Reset"; taps .VRD01.CLIM.InitOK
button at (10,10)-(71,41): text "Home"; opens PLC_VISU
rectangle at (80,250)-(221,271): text "T-Set = %.1f °C"; shows INT_TO_REAL(.VRD01.SetPoint)/10
rectangle at (270,60)-(431,81): text "Climatica VRD02"
button at (430,60)-(471,81): text "Reset"; taps .VRD02.CLIM.InitOK; runs INTERN ASSIGN VRD02_Clima.InitOK:=(FALSE)
rectangle at (310,250)-(451,271): text "T-Set = %.1f °C"; shows INT_TO_REAL(.VRD02.SetPoint)/10
rectangle at (40,230)-(91,251): text "%.1f °C"; shows INT_TO_REAL(.TPV04.IN)/10
rectangle at (270,230)-(321,251): text "%.1f °C"; shows INT_TO_REAL(.TPV05.IN)/10
rectangle at (570,60)-(731,81): text "Climatica CAL01"
button at (730,60)-(771,81): text "Reset"; taps .VRD02.CLIM.InitOK; runs INTERN ASSIGN VRD02_Clima.InitOK:=(FALSE)
rectangle at (620,260)-(761,281): text "T-Set = %.1f °C"; shows INT_TO_REAL(.CAL01.SetPoint)/10
rectangle at (80,10)-(781,41): text "%s"; shows .Plant_NAME
rectangle at (40,330)-(201,351): text "Climatica VRD03"
button at (200,330)-(241,351): text "Reset"; taps .VRD03.CLIM.InitOK; runs INTERN ASSIGN VRD02_Clima.InitOK:=(FALSE)
rectangle at (70,520)-(211,541): text "T-Set = %.1f °C"; shows INT_TO_REAL(.VRD03.Ctrl_SetPoint)/10
rectangle at (40,500)-(91,521): text "%.1f °C"; shows INT_TO_REAL(.TPV06.IN)/10
rectangle at (600,300)-(761,321): text "k Scambiatore = %.1f °C"; shows INT_TO_REAL(.OffsetSetPointManuale/10)
rectangle at (280,330)-(441,351): text "Climatica VRD04"
button at (440,330)-(481,351): text "Reset"; taps .VRD04.CLIM.InitOK; runs INTERN ASSIGN VRD02_Clima.InitOK:=(FALSE)
rectangle at (270,520)-(391,541): text "T-Set = %.1f °C"; shows INT_TO_REAL(.VRD04.SetPoint)/10
rectangle at (280,500)-(331,521): text "%.1f °C"; shows INT_TO_REAL(.TPV06.IN)/10
rectangle at (190,230)-(251,251): text "MAN"; invisible if NOT .VRD01.ComandoManuale
rectangle at (420,230)-(481,251): text "MAN"; invisible if NOT .VRD02.ComandoManuale
rectangle at (190,500)-(251,521): text "MAN"; invisible if NOT .VRD03.ComandoManuale
rectangle at (430,500)-(491,521): text "MAN"; invisible if NOT .VRD04.ComandoManuale
rectangle at (600,320)-(761,341): text "k Scambiatore 2 = %.1f °C"; shows INT_TO_REAL(.OffsetSetPointManuale2/10)
rectangle at (610,460)-(791,481): text "Offset Boost = %.1f °C"; shows INT_TO_REAL(.RifOffsetBoost/10)
rectangle at (610,480)-(791,501): text "Boost Attivo"; invisible if NOT .BitAbilitaBoost
rectangle at (610,480)-(791,501): text "Boost NON Attivo"; invisible if .BitAbilitaBoost
rectangle at (10,320)-(261,591): text "( * VRD03 Esclusa perchè bypassata * )"
rectangle at (610,510)-(791,531): text "Soglia Start Antigelo = %.1f °C"; shows INT_TO_REAL((.SogliaMinStartAntigelo)/10)
rectangle at (610,550)-(791,571): text "Antigleo Attivo"; invisible if NOT .PLC_PRG.StartCAL_Antigelo.Q1
rectangle at (610,550)-(791,571): text "Antigelo NON Attivo"; invisible if .PLC_PRG.StartCAL_Antigelo.Q1
rectangle at (610,530)-(791,551): text "Soglia Stop Antigelo = %.1f °C"; shows INT_TO_REAL((.SogliaMinStopAntigelo)/10)
rectangle at (590,340)-(761,361): text "T_S01 Esterna  = %.1f °C"; shows INT_TO_REAL(.TPV01.IN)/10
rectangle at (600,280)-(761,301): text "T_S02 Mandata  = %.1f °C"; shows INT_TO_REAL(.TPV02.AVG)/10
rectangle at (550,370)-(771,391): text "Correzione Set Point VRD04"
rectangle at (550,390)-(661,411): text "T_S08  = %.1f °C"; shows INT_TO_REAL(.TPV08.IN)/10
rectangle at (680,390)-(791,411): text "Offset = %.1f °C"; shows INT_TO_REAL(PLC_PRG.OffsetVRD04)/10
6 more shapes without text or variables
81 elements of other kinds (tables, trends, ...) not read
*)
